METHOD PROTECTED getValue : BOOL //Return value = TRUE if execution finished and state incremented 
VAR_INPUT
	Index						:	WORD;
	SubIndex					:	BYTE;
	Len							:	UDINT;
	pActValue					:	PVOID; //Address of variable for actual value
	pSetValue					:	PVOID; //Address of variable for ser value variable, can be zero if no corresponding SetVariable exists
	CompleteAccess				:	BOOL;
END_VAR
CoERead(bExecute := TRUE , nIndex := Index ,nSubIndex := SubIndex ,pDstBuf := pActValue ,cbBufLen := Len, bCompleteAccess  := CompleteAccess);
IF NOT CoERead.bBUSY 	
THEN
	IF NOT CoERead.bError
	THEN
		IF pSetValue <> 0 THEN MEMCPY(pSetValue, pActValue, Len); END_IF
		state 												:= state + 1; 
	ELSE
		Busy												:= FALSE;
		Error												:= TRUE;
		ErrorId												:= CoERead.nErrId;
		ErrorText											:= CONCAT('Error read parameter in state:' , TO_STRING(state * -1));
		ErrorText											:= CONCAT(ErrorText , ' Id:');
		ErrorText											:= CONCAT(ErrorText , TO_STRING(ErrorId));
		State												:= 9999;
	END_IF
	CoERead(bExecute := FALSE);
	getValue												:= TRUE;
END_IF
END_METHOD

METHOD PROTECTED seqRead : BOOL //Return value = TRUE if execution finished 
VAR_IN_OUT
	State							:	INT;
END_VAR

(* Sequence read parameter **********************************)
	CASE state OF
	1..99: //Read application specific parameter  
		seqRead												:= TRUE;
		
	1001: (* Init step ******************************************************)
		CoERead(bExecute := FALSE, sNetId:= F_CreateAmsNetId(nIds := AdsAddr.netId), nSlaveAddr:= AdsAddr.port);
		IF NOT CoERead.bBusy
		THEN
			state											:= state + 1;	
		END_IF
		
	1002: (* Device name *************************************************************************************)
		IF LEN(DeviceType) > 0 AND NOT CoERead.bBusy
		THEN
			state											:= state + 1;
		ELSE
			getValue(Index:= 16#1008,	Subindex := 16#0,	LEN := SIZEOF(DeviceType),	pActValue := ADR(DeviceType),	pSetValue := 0, completeAccess := FALSE);
		END_IF

			
	1003: (* kp_current *************************************************************************************)
		IF DeviceType = 'EL7041-1000' OR DeviceType = 'EP7041-3002' OR DeviceType = 'EP7041-3102'
		THEN
			state											:= state + 1; (* NOT available *)
		ELSE	
			IF getValue(Index:= 16#8011,	Subindex := 16#01,	LEN := SIZEOF(_UINT),	pActValue := ADR(_UINT),	pSetValue := 0, completeAccess := FALSE)
			THEN
				KpCurrent := SetKpCurrent					:= SEL(Error, UINT_TO_LREAL(_UINT), 0.0);
			END_IF
		END_IF
		
	1004: (* ki current **********************************)
		IF DeviceType = 'EL7041-1000' OR DeviceType = 'EP7041-3002' OR DeviceType = 'EP7041-3102'
		THEN
			state											:= state + 1; (* Not available *)
		ELSE	
			IF getValue(Index:= 16#8011,	Subindex := 16#02,	LEN := SIZEOF(_UINT),	pActValue := ADR(_UINT),	pSetValue := 0, completeAccess := FALSE)
			THEN
				KiCurrent := SetKiCurrent					:= SEL(Error, UINT_TO_LREAL(_UINT), 0.0);
			END_IF		
		END_IF
	
	1005: (* Kp velocity ****************************************************************************************)
		IF DeviceType = 'EL7041-1000'
		THEN
			state											:= state + 1;
		ELSIF DeviceType = 'EL7037' OR DeviceType = 'EL7047' 
		THEN			
			IF getValue(Index:= 16#8014,	Subindex := 16#03,	LEN := SIZEOF(_UDINT),	pActValue := ADR(_UDINT),	pSetValue := 0, completeAccess := FALSE)
			THEN
				KpVelocity := SetKpVelocity					:= SEL(Error, UDINT_TO_LREAL(_UDINT), 0.0);
			END_IF
		ELSE			
			IF getValue(Index:= 16#8013,	Subindex := 16#01,	LEN := SIZEOF(_UINT),	pActValue := ADR(_UINT),	pSetValue := 0, completeAccess := FALSE)
			THEN
				KpVelocity := SetKpVelocity					:= SEL(Error, UINT_TO_LREAL(_UINT), 0.0);
			END_IF			
		END_IF	
		
	1006: (* Tn velocity or Ki Velocity ****************************************************************************************)
		IF DeviceType = 'EL7041-1000'
		THEN
			state											:= state + 1;
		ELSIF DeviceType = 'EL7037' OR DeviceType = 'EL7047'
		THEN (* Tn velocity*)			
			IF getValue(Index:= 16#8014,	Subindex := 16#04,	LEN := SIZEOF(_UINT),	pActValue := ADR(_UINT),	pSetValue := 0, completeAccess := FALSE)
			THEN
				KiVelocity := SetKiVelocity					:= SEL(Error, UINT_TO_LREAL(_UINT), 0.0);
			END_IF
			
		ELSE (* Ki Velccity*)
			IF getValue(Index:= 16#8013,	Subindex := 16#02,	LEN := SIZEOF(_UINT),	pActValue := ADR(_UINT),	pSetValue := 0, completeAccess := FALSE)
			THEN
				KiVelocity := SetKiVelocity					:= SEL(Error, UINT_TO_LREAL(_UINT), 0.0);
			END_IF
		END_IF 
	
	1007: (* Kp position ****************************************************************************************)
		IF DeviceType = 'EL7037' OR DeviceType = 'EL7047' 
		THEN			
			IF getValue(Index:= 16#8014,	Subindex := 16#02,	LEN := SIZEOF(_UINT),	pActValue := ADR(_UINT),	pSetValue := 0, completeAccess := FALSE)
			THEN
				KpPosition := SetKpPosition					:= SEL(Error, UINT_TO_LREAL(_UINT), 0.0);
			END_IF			
		ELSE
			;
		END_IF	
	
	1008: (* Homing cam search direction ****************************************************************************************)		
		IF DeviceType = 'EL7041-1000' 
		THEN
			state											:= state + 1;
		ELSE
			getValue(Index:= 16#8021,	Subindex := 16#13,	LEN := SIZEOF(CalibrInvertDirForCamSearch),	pActValue := ADR(CalibrInvertDirForCamSearch),	pSetValue := ADR(SetCalibrInvertDirForCamSearch), completeAccess := FALSE);			
		END_IF
	
	1009: (* Homing cam of direxction ****************************************************************************************)	
		IF DeviceType = 'EL7041-1000'
		THEN
			state											:= state + 1;
		ELSE
			getValue(Index:= 16#8021,	Subindex := 16#14,	LEN := SIZEOF(CalibrInvertDirForOfCam),	pActValue := ADR(CalibrInvertDirForOfCam),	pSetValue := ADR(SetCalibrInvertDirForOfCam), completeAccess := FALSE);			
		END_IF

	1010: (* Calibration value ****************************************************************************************)
		IF DeviceType = 'EL7041-1000'
		THEN
			state											:= state + 1;
		ELSE
			getValue(Index:= 16#8020,	Subindex := 16#08,	LEN := SIZEOF(CalibrPosition),	pActValue := ADR(CalibrPosition),	pSetValue := ADR(SetCalibrPosition), completeAccess := FALSE);			
		END_IF
		
	ELSE
		state												:= 1;
	END_CASE

(***********************************************************************************)
END_METHOD

METHOD PROTECTED seqWrite : BOOL //Return value = TRUE if execution finished 
VAR_IN_OUT
	State							:	INT;
END_VAR

(* Sequence write parameter *********************************************)
	CASE state OF
	1..99: //Write application specific parameter  
		seqWrite											:= TRUE;
		
	1001: (* Init step ******************************************************)
		CoEWrite(bExecute := FALSE, sNetId:= F_CreateAmsNetId(nIds := AdsAddr.netId), nSlaveAddr:= AdsAddr.port);
		IF NOT CoEWrite.bBusy
		THEN
			state											:= state + 1;	
		END_IF
		
	1002: (* Kv position *************************************************************************************)
		IF DeviceType = 'EL7041-1000' OR DeviceType = 'EP7041-3002' OR DeviceType = 'EP7041-3102'
			OR KpCurrent = SetKpCurrent AND NOT CoEWrite.bBusy
		THEN
			state											:= state + 1;
		ELSE
			_UINT											:= LREAL_TO_UINT(SetKpCurrent);
			IF setValue(Index:= 16#8011,	Subindex := 16#01,	LEN := SIZEOF(_UINT),		pActValue := 0,		pSetValue := ADR(_UINT) , completeAccess := FALSE)
			THEN
				KpCurrent									:= SetKpCurrent;
			END_IF			
		END_IF	
		
	1003: (* ki current **********************************)
		IF DeviceType = 'EL7041-1000' OR DeviceType = 'EP7041-3002' OR DeviceType = 'EP7041-3102'
			OR KiCurrent = SetKiCurrent AND NOT CoEWrite.bBusy
		THEN
			state											:= state + 1;
		ELSE
			_UINT											:= LREAL_TO_UINT(SetKiCurrent);
			IF setValue(Index:= 16#8011,	Subindex := 16#02,	LEN := SIZEOF(_UINT),		pActValue := 0,		pSetValue := ADR(_UINT) , completeAccess := FALSE)
			THEN
				KiCurrent									:= SetKiCurrent;
			END_IF			
		END_IF
	
	1004: (* Kp velocity ****************************************************************************************)
		IF DeviceType = 'EL7041-1000' 
			OR KpVelocity = SetKpVelocity AND NOT CoEWrite.bBusy
		THEN
			state											:= state + 1;
		ELSE
			IF DeviceType = 'EL7037' OR DeviceType = 'EL7047' 
			THEN
				_UDINT										:=LREAL_TO_UDINT(SetKpVelocity);
				IF setValue(Index:= 16#8014,	Subindex := 16#03,	LEN := SIZEOF(_UDINT),		pActValue := 0,		pSetValue := ADR(_UDINT) , completeAccess := FALSE)
				THEN
					KpVelocity								:= SetKpVelocity;
				END_IF	
			ELSE
				_UINT										:=LREAL_TO_UINT(SetKpVelocity);
				IF setValue(Index:= 16#8013,	Subindex := 16#01,	LEN := SIZEOF(_UINT),		pActValue := 0,		pSetValue := ADR(_UINT) , completeAccess := FALSE)
				THEN
					KpVelocity								:= SetKpVelocity;
				END_IF	
			END_IF		
		END_IF
	
	1005: (* Tn velocity or Ki velocity****************************************************************************************)
		IF SetTnVelocity = TnVelocity AND SetKiVelocity = KiVelocity AND NOT CoEWrite.bBusy OR DeviceType = 'EL7041-1000'
		THEN 
			state											:= state + 1;
		ELSE
			IF DeviceType = 'EL7037' OR DeviceType = 'EL7047' 
			THEN (* Tn Velocity *)
				_UINT										:= LREAL_TO_UINT(SetTnVelocity);
				IF setValue(Index:= 16#8014,	Subindex := 16#04,	LEN := SIZEOF(_UINT),		pActValue := 0,		pSetValue := ADR(_UINT) , completeAccess := FALSE)
				THEN
					TnVelocity								:= SetTnVelocity;
				END_IF	
				
	
			ELSE (* Ki Velocity *)
				_UINT										:= LREAL_TO_UINT(SetKiVelocity);
				IF setValue(Index:= 16#8013,	Subindex := 16#02,	LEN := SIZEOF(_UINT),		pActValue := 0,		pSetValue := ADR(_UINT) , completeAccess := FALSE)
				THEN
					KiVelocity								:= SetKiVelocity;
				END_IF				
			END_IF	
		END_IF
	
	1006: (* Kp position ****************************************************************************************)		
		IF SetKpPosition <> KpPosition AND (DeviceType = 'EL7037' OR DeviceType = 'EL7047')
		THEN
			_UINT											:= LREAL_TO_UINT(SetKpPosition);
			IF setValue(Index:= 16#8014,	Subindex := 16#02,	LEN := SIZEOF(_UINT),		pActValue := 0 ,		pSetValue := ADR(_UINT) , completeAccess := FALSE)	
			THEN
				KpPosition									:= SetKpPosition;
			END_IF			
		ELSIF NOT CoEWrite.bBusy
		THEN
			state											:= state + 1;
		END_IF
			
	1007: (* Homing cam search direction ********************************************************************************************)
		IF DeviceType = 'EL7041-1000' 
		THEN
			state											:= state + 1;
		ELSE
			setValue(Index:= 16#8021,	Subindex := 16#13,	LEN := SIZEOF(SetCalibrInvertDirForCamSearch),		pActValue := ADR(CalibrInvertDirForCamSearch) ,		pSetValue := ADR(SetCalibrInvertDirForCamSearch) , completeAccess := FALSE);
		END_IF
		
	1008: (* Homing cam of direction *****************************************************************************************)
		IF DeviceType = 'EL7041-1000' 
		THEN
			state											:= state + 1;
		ELSE
			setValue(Index:= 16#8021,	Subindex := 16#14,	LEN := SIZEOF(SetCalibrInvertDirForOfCam),		pActValue := ADR(CalibrInvertDirForOfCam) ,		pSetValue := ADR(SetCalibrInvertDirForOfCam) , completeAccess := FALSE)	;	
		END_IF
	
	1009: (* Calibration position ***********************************************************************)	
		IF DeviceType = 'EL7041-1000' 
		THEN
			state											:= state + 1;
		ELSE
			setValue(Index:= 16#8020,	Subindex := 16#08,	LEN := SIZEOF(SetCalibrPosition),		pActValue := ADR(CalibrPosition) ,		pSetValue := ADR(SetCalibrPosition) , completeAccess := FALSE)	;	
		END_IF
	ELSE
		state												:= 1;
	END_CASE

(************************************************************************************)
END_METHOD

METHOD PROTECTED setValue : BOOL //Return value = TRUE if execution finished and state incremented 
VAR_INPUT
	Index						:	Word;
	SubIndex					:	BYTE;
	Len							:	UDINT;
	pActValue					:	PVOID; //Address of variable for actual value, can be zero if no corresponding acual value variable exists
	pSetValue					:	PVOID; //Address of variable for set value variable
	CompleteAccess				:	BOOL;
END_VAR


IF pActValue <> 0 AND pSetValue <> 0 AND_THEN MEMCMP(pSetValue, pActValue, Len) = 0
THEN //Skip write parameter if set and actual value are equel
	state													:= state + 1;	
	setValue												:= TRUE;
ELSE
	CoEWrite(bExecute := TRUE, nIndex := Index ,nSubIndex := SubIndex , pSrcBuf := pSetValue ,cbBufLen := Len , bCompleteAccess := CompleteAccess );
	IF NOT CoEWrite.bBusy
	THEN
		IF NOT CoEWrite.bError
		THEN
			IF pActValue <> 0 THEN MEMCPY(pActValue, pSetValue, Len); END_IF	
			state											:= state + 1;
		ELSE
			Busy											:= FALSE;
			Error											:= TRUE;
			ErrorId											:= CoEWrite.nErrId;
			ErrorText										:= CONCAT('Error write parameter in state:' , TO_STRING(state * -1));
			ErrorText										:= CONCAT(ErrorText , ' Id:');
			ErrorText										:= CONCAT(ErrorText , TO_STRING(ErrorId));
			State											:= 9999;
		END_IF
		CoEWrite(bExecute := FALSE);
		setValue											:= TRUE;
	END_IF		
END_IF
END_METHOD

END_FUNCTION_BLOCK

// POUs/IO/Drives/AxDriveGetRef
{attribute 'no_check'}
//Provides drive reference (Ref -> ST_DriveRef) based on NC-AxisID
//Drive reference is needed for FB's of lib Drive e.g. FB_SoEAX5000FirmwareUpdate_ByDriveRef
FUNCTION_BLOCK AxDriveGetRef EXTENDS FbBase
VAR CONSTANT                								
	NCIDXG_AXPARMS											: UDINT := 16#0000_4000;	(* Axis with ID: Parameter 			*)
	NCIDXO_AXP_HWAMSADDR									: UDINT := 16#0000_0031;	
	MIN_ADSREAD_BUFFER										:	INT := 0;
	MAX_ADSREAD_BUFFER										:	INT := 9;
END_VAR 
VAR_INPUT                   					
	AmsNetId												: T_AmsNetId := '';	(* netID of PC with NC *)			      
	AxisId													:	DWORD; //NC axis id	
END_VAR
VAR_OUTPUT                  								
	DriveAmsNetId											: T_AmsNetIdArr; (* Ams net id as array of bytes *)
    DriveRef												: ST_DriveRef; 	(* contains sNetID of EcMaster, nSlaveAddr of EcDrive, nDriveNo of EcDrive, either preset or read from NC *)
END_VAR              								                 								
VAR                         								
(* cache ********************************************)
	AdsReadBuffer											: ARRAY[MIN_ADSREAD_BUFFER..MAX_ADSREAD_BUFFER] OF BYTE;
                						
(* trigger ******************************************)

(* timer ********************************************)
	
(* blocks *******************************************)	
	AdsRead													: ADSREAD := (TMOUT := DEFAULT_ADS_TIMEOUT);
	
(* dummys *******************************************)
END_VAR

	(* Create drive ref for device 									*)
	(****************************************************************)

(* Sequence ****************************************)
	rtExecute(CLK := Execute);
	CASE state OF 
	0:	
		Busy												:= FALSE;
		IF NOT Execute
		THEN
			Done											:= FALSE;
			Error											:= FALSE;
			ErrorId											:= 0;
		ELSIF rtExecute.Q
		THEN
			Busy											:= TRUE;
			Done											:= FALSE;
			Error											:= FALSE;
			ErrorId											:= 0;
			AdsRead(READ := FALSE);
			MEMSET(ADR(DriveRef), 0, SIZEOF(DriveRef));
			MEMSET(ADR(AdsReadBuffer), 0, SIZEOF(AdsReadBuffer));
			state											:= State + 1;
		END_IF 
	
	1: //Get drive slave address
		AdsRead(
			NETID	:= AmsNetId,
			PORT	:= AMSPORT_R0_NC,
			IDXGRP	:= NCIDXG_AXPARMS + AxisId,
			IDXOFFS	:= NCIDXO_AXP_HWAMSADDR,
			LEN		:= SIZEOF(AdsReadBuffer) ,
			DESTADDR:= ADR(AdsReadBuffer),
			READ	:= TRUE);
		IF NOT AdsRead.BUSY
		THEN
			IF NOT AdsRead.ERR 
			THEN
				MEMCPY(ADR(DriveAmsNetId), ADR(AdsReadBuffer), SIZEOF(DriveAmsNetId)); 							(* AdsreadBuffer[0..5] *)
				MEMCPY(ADR(DriveRef.nSlaveAddr), ADR(AdsReadBuffer[6]), SIZEOF(DriveRef.nSlaveAddr));  	(* AdsreadBuffer[6..7] *)
				MEMCPY(ADR(DriveRef.nDriveNo), ADR(AdsReadBuffer[8]), SIZEOF(DriveRef.nDriveNo));  		(* AdsreadBuffer[8..9] *)

				(* create string out of byte array *)
				DriveRef.sNetId 							:= F_CreateAmsNetId(DriveAmsNetId);
				
				Busy										:= FALSE;
				Done										:= TRUE;
				state										:= 0;
			ELSE
				Busy										:= FALSE;
				Error										:= TRUE;
				ErrorId										:= AdsRead.ERRID;
				State										:= 0;
			END_IF
		END_IF
	END_CASE
	
(**********************************************************************************)

END_FUNCTION_BLOCK

// POUs/IO/EL-EP/EL3403/EL3403
{attribute 'no_check'}
FUNCTION_BLOCK EL3403 Extends EcSlaveInfoData
VAR CONSTANT
	MIN_PHASE												:	INT := 1;
	MAX_PHASE												:	INT := 3;
END_VAR  
VAR_INPUT
	IndexOut										AT %Q*	:	ARRAY[MIN_PHASE..MAX_PHASE] OF USINT;
	Transmission											:	ARRAY[MIN_PHASE..MAX_PHASE] OF LREAL;	//Transmission current transformator for each phase e.g. 750 *)
END_VAR
VAR_OUTPUT
	(* Inputs Channel 1-3 *)
	TxPDOToggle										AT %I*	: 	ARRAY[MIN_PHASE..MAX_PHASE] OF BOOL;
	IndexIn											AT %I*	: 	ARRAY[MIN_PHASE..MAX_PHASE] OF USINT;
	Current													: 	ARRAY[MIN_PHASE..MAX_PHASE] OF LREAL; 	//Unit: 0,000001 A
	Voltage													: 	ARRAY[MIN_PHASE..MAX_PHASE] OF LREAL; 	//Unit: 0,0001 V
	ActivePower												: 	ARRAY[MIN_PHASE..MAX_PHASE] OF LREAL; 	//Unit: 0,01 W

	(* PM Status Data *)
	MissingZeroCrossingA							AT %I*	: 	BOOL;
	MissingZeroCrossingB							AT %I* 	: 	BOOL;
	MissingZeroCrossingC							AT %I* 	: 	BOOL;
	PhaseSequenceError								AT %I* 	: 	BOOL;
//	SyncError										AT %I* 	: 	BOOL;
                                                              	
	(* MultiplexValues	*)
	ApparentPower											:	ARRAY[MIN_PHASE..MAX_PHASE] OF LREAL; 	//apparent power unit: 0,01 VA
	ReactivePower											:	ARRAY[MIN_PHASE..MAX_PHASE] OF LREAL; 	//reactive power unit: 0,01 VAr
	PowerFactor												:	ARRAY[MIN_PHASE..MAX_PHASE] OF LREAL; 	//effective power cos phi Unit: 0,001
	EnergyConsumption										:	ARRAY[MIN_PHASE..MAX_PHASE] OF LREAL; 	//energy unit: 0,001 Wh
	EnergyConsumptionInvers									:	ARRAY[MIN_PHASE..MAX_PHASE] OF LREAL; 	//energy unit: 0,001 Wh
	TimestampDistClocks										:	ARRAY[MIN_PHASE..MAX_PHASE] OF LREAL; 	//timestamp unit : 1 ns
	Frequency												:	ARRAY[MIN_PHASE..MAX_PHASE] OF LREAL; 	//frequenzy unit : 0,1 Hz

END_VAR
VAR (* Internal IOs *)
	_Current										AT %I* 	: 	ARRAY[MIN_PHASE..MAX_PHASE] OF DINT; 	//Unit: 0,000001 A
	_Voltage										AT %I* 	: 	ARRAY[MIN_PHASE..MAX_PHASE] OF DINT; 	//Unit: 0,0001 V
	_ActivePower									AT %I* 	: 	ARRAY[MIN_PHASE..MAX_PHASE] OF DINT; 	//Unit: 0,01 W

	_VariantValue									AT %I* 	: 	ARRAY[MIN_PHASE..MAX_PHASE] OF DINT;
//	_SyncErrorChannel								AT %I* 	: 	ARRAY[MIN_PHASE..MAX_PHASE] OF BOOL; 	//reserved
//	_SyncErrorTerminal										: 	BOOL;	//reserved
END_VAR                       							
VAR
	i														:	INT;
END_VAR

(* EL 3403 IO 									*)
(************************************************)

(* Get Index Values *****************************)
	FOR i := MIN_PHASE TO MAX_PHASE DO
		Current[i]											:= Transmission[i] * DINT_TO_LREAL(_Current[i]) / 1000000.0; //A
		Voltage[i]											:= (*Uebersetzung[i] **) DINT_TO_LREAL(_Voltage[i]) / 10000.0; //V
		ActivePower[i]										:= Transmission[i] * DINT_TO_LREAL(_ActivePower[i]) / 100.0; //W
                                            				
		CASE IndexIn[i] OF                  				
		0:(*Scheinleistung*)                				
			ApparentPower[i]								:= Transmission[i] * DINT_TO_LREAL(_VariantValue[i]) / 100.0; //VA
                                            				
		1:(*Blindleistung*)                 				
			ReactivePower[i]								:= Transmission[i] * DINT_TO_LREAL(_VariantValue[i]) / 100.0; //VAr
                                            				
		2:(*Energie*)                       				
			EnergyConsumption[i]							:= Transmission[i] * DINT_TO_LREAL(_VariantValue[i]) / 1000.0; //Wh
                                            				
		3:(*Wirkleistungsfaktor*)           				
			PowerFactor[i]									:= DINT_TO_LREAL(_VariantValue[i]) / 1000.0; //cos phi
                                            				
		4:(*Frequenz*)                      	
			Frequency[i]									:= DINT_TO_LREAL(_VariantValue[i]) / 10.0; //Hz
                                            				
		5:(*Energie Invers*)                				
			EnergyConsumptionInvers[i]						:= Transmission[i] * DINT_TO_LREAL(_VariantValue[i]) / 1000.0;
                                            				
		100:(*Zeitstempel*)                 				
			TimestampDistClocks[i]							:= DINT_TO_LREAL(_VariantValue[i]);
	
		END_CASE

	END_FOR

(***********************************************)

END_FUNCTION_BLOCK

// POUs/IO/EL-EP/EL3403/EL3403Logic
{attribute 'no_check'}
//FB gets raw data from EL3404 every cycle and calculate real values *)
FUNCTION_BLOCK EL3403Logic
VAR_INPUT
	TrigReadVariantValues									:	BOOL 	:= FALSE;	//Rising edge reports actual total values on FB outputs
	Transmission											:	LREAL 	:= 750.0; 	//Transmission current transformator
	Mode													:	INT 	:= 0; 		(* 	0 = Phase 1-3
																					  	1 = Phase 1
																					 	2 = Phase 2
																					 	3 = Phase 3 *)                                   						
END_VAR                             	
VAR_OUTPUT
	(* Components OUTPUT -> ReadOnly ! *)
	IO														:	EL3403;
                                    				                                					
	(* Total Values *)              					
	TotalEffectivePower										: 	LREAL; 	//W
	TotalPowerFactor										: 	LREAL; 	//total power factor cos phi
	TotalEnergyConsumption									: 	LREAL; 	//Wh
                                    					
	(* Error *)                     					
	ErrorPhaseSequence										:	BOOL;
	ErrorMissingZeroCrossing								:	BOOL;
	TimeStart												: 	TIME;		(* Startzeit *)
	TimeEnd													: 	TIME;		(* Endzeit *)
	TimeDiff												: 	TIME;		(* Differenz Start End *)
	
	(* Ctrl Status  *)              					
	Valid													:	BOOL;	//TRUE when data is valid
	Busy													:	BOOL;	//Busy is TRUE at the rising edge of Execute and FALSE when one of the outputs Done, Aborted, or Error is set 
	Error													:	BOOL;	//Rising edge of Error informs that an error occurred during the execution of the Function Block 

END_VAR                             	
VAR                                 	
	rtReadVariantValues										:	R_Trig;
	state													:	INT;
	_MIN_PHASE												:	INT;
	_MAX_PHASE												:	INT;
	i														:	INT;
END_VAR

(* Work EL3403 data 						*)
(********************************************)

(* Work Termianl IO ******************************************)
	FOR i := IO.MIN_PHASE TO IO.MAX_PHASE 
	DO
		IO.Transmission[i] 									:= Transmission;
	END_FOR

	IO();

(* Error *****************************************************)
	Error 													:= IO.WCState OR IO.InfoDataState <> Tc2_EtherCAT.EC_DEVICE_STATE_OP;

(* Get Total Values ******************************************)
IF NOT Error
THEN
	CASE Mode OF
	1:
		TotalEffectivePower 								:= IO.ActivePower[1];
		TotalPowerFactor 									:= IO.PowerFactor[1];
		TotalEnergyConsumption 								:= IO.EnergyConsumption[1];
	2:                              						
		TotalEffectivePower 								:= IO.ActivePower[2];
		TotalPowerFactor 									:= IO.PowerFactor[2];
		TotalEnergyConsumption 								:= IO.EnergyConsumption[2];
	3:                              						
		TotalEffectivePower 								:= IO.ActivePower[3];
		TotalPowerFactor 									:= IO.PowerFactor[3];
		TotalEnergyConsumption 								:= IO.EnergyConsumption[3];
	ELSE (* Phase 1-3 *)            						
		TotalEffectivePower 								:= IO.ActivePower[1] + IO.ActivePower[2] + IO.ActivePower[3];
		TotalPowerFactor 									:= (IO.PowerFactor[1] + IO.PowerFactor[2] + IO.PowerFactor[3]) / 3.0;
		TotalEnergyConsumption 								:= IO.EnergyConsumption[1] + IO.EnergyConsumption[2] + IO.EnergyConsumption[3];
	END_CASE                        	

END_IF

(* Trigger ReadVariantValues ******************************)
rtReadVariantValues(CLK := TrigReadVariantValues);

IF rtReadVariantValues.Q
	OR state <> 0
THEN
	ReadVariantValues(Mode := Mode);
END_IF

(********************************************************)

METHOD PUBLIC readVariantValues : Bool //Return value = TRUE if busy
VAR_INPUT
	Mode								:	INT 	:= 0; (* 	0 = Phase 1-3
															  		1 = Phase 1
															 	 	2 = Phase 2
															 		3 = Phase 3 *)
END_VAR
IF state = 0 
THEN
	THIS^.Mode												:= Mode;
	CASE mode OF
	1:
		_MIN_PHASE 											:= IO.MIN_PHASE;
		_MAX_PHASE 											:= IO.MIN_PHASE;
	2:             											
		_MIN_PHASE 											:= IO.MIN_PHASE + 1;
		_MAX_PHASE 											:= IO.MIN_PHASE + 1;
	3:             											
		_MIN_PHASE 											:= IO.MAX_PHASE;
		_MAX_PHASE 											:= IO.MAX_PHASE;
	ELSE           											
		_MIN_PHASE 											:= IO.MIN_PHASE;
		_MAX_PHASE 											:= IO.MAX_PHASE;
	END_CASE
	state 													:= 1;
	TimeStart 												:= TIME();
END_IF

(* Read Variant Values *******************************)
	CASE state OF
	0:
		;
		
	1:
		FOR i := _MIN_PHASE TO _MAX_PHASE DO
			IO.IndexOut[i] 									:= 0;
			IF IO.IndexIn[i] = IO.IndexOut[i]
				AND i = _MAX_PHASE
			THEN (* Set Next index *)
				state 										:= 2;
			ELSE
				;
			END_IF
		END_FOR

	2:
		FOR i := _MIN_PHASE TO _MAX_PHASE DO
			IO.IndexOut[i] 									:= 1;
			IF IO.IndexIn[i] = IO.IndexOut[i]
				AND i = _MAX_PHASE
			THEN (* Set Next index *)
				state 										:= 3;
			ELSE
				;
			END_IF
		END_FOR
	3:
		FOR i := _MIN_PHASE TO _MAX_PHASE DO
			IO.IndexOut[i] 									:= 2;
			IF IO.IndexIn[i] = IO.IndexOut[i]
				AND i = _MAX_PHASE
			THEN (* Set Next index *)
				state 										:= 4;
			ELSE
				;
			END_IF
		END_FOR
	4:
		FOR i := _MIN_PHASE TO _MAX_PHASE DO
			IO.IndexOut[i] 									:= 3;
			IF IO.IndexIn[i] = IO.IndexOut[i]
				AND i = _MAX_PHASE
			THEN (* Set Next index *)
				state 										:= 5;
			ELSE
				;
			END_IF
		END_FOR
	5:
		FOR i := _MIN_PHASE TO _MAX_PHASE DO
			IO.IndexOut[i] 									:= 4;
			IF IO.IndexIn[i] = IO.IndexOut[i]
				AND i = _MAX_PHASE
			THEN (* Set Next index *)
				state 										:= 6;
			ELSE
				;
			END_IF
		END_FOR

	6:
		FOR i := _MIN_PHASE TO _MAX_PHASE DO
			IO.IndexOut[i] 									:= 5;
			IF IO.IndexIn[i] = IO.IndexOut[i]
				AND i = _MAX_PHASE
			THEN (* Set Next index *)
				state 										:= 7;
			ELSE
				;
			END_IF
		END_FOR

	7:
		FOR i := _MIN_PHASE TO _MAX_PHASE DO
			IO.IndexOut[i] 									:= 100;
			IF IO.IndexIn[i] = IO.IndexOut[i]
				AND i = _MAX_PHASE
			THEN (* Set Next index *)
				Valid 										:= TRUE;
				state 										:= 0;
				TimeEnd 									:= TIME();
				TimeDiff 									:= TimeEnd - TimeStart;
			ELSE
				;
			END_IF
		END_FOR

	END_CASE
	
	Busy													:= state <> 0;
	ReadVariantValues 										:= Busy;
END_METHOD

END_FUNCTION_BLOCK

// POUs/IO/EL-EP/EL9x/EL95xxPowerTerminal
{attribute 'no_check'}
FUNCTION_BLOCK EL95xxPowerTerminal 
VAR_OUTPUT CONSTANT
END_VAR
VAR_INPUT
END_VAR
VAR_OUTPUT	
	PowerOK			 									AT  %I* : BOOL;
	Overload											AT  %I* : BOOL;
END_VAR
VAR
END_VAR

	(* EL95xx Power supply terminal			*)
	(****************************************)
	
(* Work objects ****************************************)
;
(*******************************************************)

END_FUNCTION_BLOCK

// POUs/IO/EL-EP/EL9x/ELSystemTerminal
{attribute 'no_check'}
FUNCTION_BLOCK ELSystemTerminal //e.g. EL9410
VAR_OUTPUT CONSTANT
END_VAR
VAR_INPUT
END_VAR
VAR_OUTPUT	
	UsUndervoltage		 								AT  %I* : BOOL;
	UpUndervoltage										AT  %I* : BOOL;
END_VAR
VAR
END_VAR

	(* System terminal power status			*)
	(****************************************)
	
(* Work objects ****************************************)
;
(*******************************************************)

END_FUNCTION_BLOCK

// POUs/IO/EL-EP/EP92xxPwrBox/EP9214
{attribute 'no_check'}
FUNCTION_BLOCK EP9214
VAR_OUTPUT CONSTANT
	MIN_CHANNEL												: INT := 1;
	MAX_CHANNEL												: INT := 4;
END_VAR
VAR_INPUT
	EnableControlViaFieldbus					AT  %Q* 	: 	BOOL := FALSE;	//FB will be processed as long as enable is TRUE
	ResetTrig									AT  %Q* 	: 	BOOL := FALSE;	//The box will be reseted with a rising edge 
	
	Channel													:	ARRAY[MIN_CHANNEL..MAX_CHANNEL] OF EP9214_CHANNEL;
END_VAR     								
VAR_OUTPUT  	
	TempWarning									AT  %I* 	: 	BOOL;	//TRUE when temperature warning occurs
	TempError									AT  %I* 	: 	BOOL;	//TRUE when temperature error occurs
	UsWarning									AT  %I* 	: 	BOOL;	//TRUE when system voltage warning occurs
	UsError										AT  %I* 	: 	BOOL;	//TRUE when system voltage error occurs
	UpWarning									AT  %I* 	: 	BOOL;	//TRUE when peripheral voltage warning occurs
	UpError										AT  %I* 	: 	BOOL;	//TRUE when peripheral voltage error occurs
	GlobalError									AT  %I* 	: 	BOOL;	//TRUE when global error occurs
	ResetInput									AT  %I* 	: 	BOOL;	//Resets box with a rising edge
	TxPDOState									AT  %I* 	: 	BOOL;	
	TxPDOToggle									AT  %I* 	: 	BOOL;	
END_VAR     								
VAR
	i														:	INT;
END_VAR

;

{attribute 'monitoring' := 'call'}
PROPERTY PUBLIC channelErrorUp : int
GET
ChannelErrorUp				:= 0;
FOR i := MIN_CHANNEL TO MAX_CHANNEL do
	IF Channel[i].ErrorUp
	THEN
		ChannelErrorUp			:= i;
		EXIT;
	END_IF	
END_FOR
END_GET
END_PROPERTY

{attribute 'monitoring' := 'call'}
PROPERTY PUBLIC channelErrorUs : int
GET
ChannelErrorUs				:= 0;
FOR i := MIN_CHANNEL TO MAX_CHANNEL do
	IF Channel[i].ErrorUs
	THEN
		ChannelErrorUs			:= i;
		EXIT;
	END_IF	
END_FOR
END_GET
END_PROPERTY

{attribute 'monitoring' := 'call'}
PROPERTY PUBLIC channelWarningUp : int
GET
ChannelWarningUp					:= 0;
FOR i := MIN_CHANNEL TO MAX_CHANNEL do
	IF Channel[i].WarningUp	
	THEN
		ChannelWarningUp			:= i;
		EXIT;
	END_IF	
END_FOR
END_GET
END_PROPERTY

{attribute 'monitoring' := 'call'}
PROPERTY PUBLIC channelWarningUs : int
GET
ChannelWarningUs					:= 0;
FOR i := MIN_CHANNEL TO MAX_CHANNEL do
	IF Channel[i].WarningUs	
	THEN
		ChannelWarningUs			:= i;
		EXIT;
	END_IF	
END_FOR
END_GET
END_PROPERTY

END_FUNCTION_BLOCK

// POUs/IO/EL-EP/EP92xxPwrBox/EP9214_CHANNEL
{attribute 'no_check'}
FUNCTION_BLOCK EP9214_CHANNEL
VAR_INPUT
	EnableUs									AT  %Q* 	: 	BOOL := TRUE; 	//switches system voltage on with a rising edge
	EnableUp									AT  %Q* 	: 	BOOL := TRUE; 	//switches peripheral voltage on with a rising edge
	ResetTrigUs	                                AT  %Q* 	: 	BOOL := FALSE;  //resets system voltage with a rising edge                    
	ResetTrigUp                                 AT  %Q* 	: 	BOOL := FALSE;	//resets peripheral voltage with a rising edge                                                                                           
END_VAR     								                          
VAR_OUTPUT  								                          
	ErrorUs										AT  %I* 	: 	BOOL := FALSE;	//TRUE when system voltage error occurs 
	ErrorUp										AT  %I* 	: 	BOOL := FALSE; 	//TRUE when peripheral voltage error occurs 
	WarningUs									AT  %I* 	: 	BOOL := FALSE; 	//TRUE when system voltage warning occurs 
	WarningUp									AT  %I* 	: 	BOOL := FALSE; 	//TRUE when peripheral voltage warning occurs 
	StatusUs									AT  %I* 	: 	BOOL := FALSE; 	//TRUE when system voltage is on
	StatusUp									AT  %I* 	: 	BOOL := FALSE; 	//TRUE when peripheral voltage is on 
	ChannelError								AT  %I* 	: 	BOOL := FALSE; 	//TRUE when channel error occurs 
	SyncError									AT  %I* 	: 	BOOL := FALSE; 	//TRUE when synchronization error occurs 
	TxPDOState									AT  %I* 	: 	BOOL := FALSE; 
	TxPDOToggle									AT  %I* 	: 	BOOL := FALSE; 
END_VAR     								
VAR
END_VAR

;

END_FUNCTION_BLOCK

// POUs/IO/EL-EP/EP92xxPwrBox/EP9224_0037
FUNCTION_BLOCK EP9224_0037
VAR_OUTPUT CONSTANT
	MIN_CHANNEL												:	INT := 1;
	MAX_CHANNEL												:	INT := 4;
END_VAR
VAR_INPUT
	EnableControlViaFieldbus					AT  %Q* 	: 	BOOL := TRUE;	// FB will be processed ads long as enable is TRUE
	ResetTrig									AT  %Q* 	: 	BOOL := FALSE;	// The box will be reseted with a rising edge 
	
	Channel													:	ARRAY[MIN_CHANNEL..MAX_CHANNEL] OF EP9224_0037_CHANNEL;
END_VAR     								
VAR_OUTPUT  
	CurrentUs									AT	%I*		:	INT;	// Actual Current Us
	CurrentUp									AT	%I*		:	INT;	// Actual Current Up
	VoltageUs									AT 	%I*		:	INT;	// Actual Voltage Us
	VoltageUp									AT 	%I*		:	INT;	// Actual Voltage Up
	Temperature									AT 	%I*		:	INT;	// Actual Temperature
	
	TempWarning												: 	BOOL;	// TRUE when temperature warning occurs
	TempError												: 	BOOL;	// TRUE when temperature error occurs
	UsWarning												: 	BOOL;	// TRUE when system voltage warning occurs
	UsError													: 	BOOL;	// TRUE when system voltage error occurs
	UpWarning												: 	BOOL;	// TRUE when peripheral voltage warning occurs
	UpError													: 	BOOL;	// TRUE when peripheral voltage error occurs
	GlobalError												: 	BOOL;	// TRUE when global error occurs
	SumCurrentWarning										:	BOOL;	// TRUE when Sum Current Warning occurs
	SumCurrentError											:	BOOL;	// True when Sum Current Error occurs
	ResetInput												: 	BOOL;	// Resets box with a rising edge
	TxPDOState												: 	BOOL;	
	TxPDOToggle												: 	BOOL;	
END_VAR     								
VAR
{attribute 'displaymode':='binary'}
	status										AT 	%I*		: 	WORD;	// Statusword
	i														:	INT;
END_VAR

FOR i := MIN_CHANNEL TO MAX_CHANNEL
DO
	Channel[i]();
END_FOR

	TempWarning			     									:= status.0;
	TempError			        								:= status.1;
	UsWarning			       								   	:= status.2;		         	     			 			
	UsError				           								:= status.3;
	UpWarning			             							:= status.4;
	UpError				           								:= status.5;
	GlobalError			    									:= status.6;
	SumCurrentWarning											:= status.7;
	SumCurrentError		     									:= status.8;
	ResetInput			     									:= status.9;
	TxPDOState			     									:= status.10;
	TxPDOToggle													:= status.11;

{attribute 'monitoring' := 'call'}
PROPERTY channelErrorUp : INT
GET
ChannelErrorUp				:= 0;
FOR i := MIN_CHANNEL TO MAX_CHANNEL do
	IF Channel[i].ErrorUp
	THEN
		ChannelErrorUp			:= i;
		EXIT;
	END_IF	
END_FOR
END_GET
END_PROPERTY

{attribute 'monitoring' := 'call'}
PROPERTY channelErrorUs : INT
GET
ChannelErrorUs				:= 0;
FOR i := MIN_CHANNEL TO MAX_CHANNEL do
	IF Channel[i].ErrorUs
	THEN
		ChannelErrorUs			:= i;
		EXIT;
	END_IF	
END_FOR
END_GET
END_PROPERTY

{attribute 'monitoring' := 'call'}
PROPERTY channelWarningUp : INT
GET
ChannelWarningUp					:= 0;
FOR i := MIN_CHANNEL TO MAX_CHANNEL do
	IF Channel[i].WarningUp
	THEN
		ChannelWarningUp			:= i;
		EXIT;
	END_IF	
END_FOR
END_GET
END_PROPERTY

{attribute 'monitoring' := 'call'}
PROPERTY channelWarningUs : INT
GET
ChannelWarningUs					:= 0;
FOR i := MIN_CHANNEL TO MAX_CHANNEL do
	IF Channel[i].WarningUs
	THEN
		ChannelWarningUs			:= i;
		EXIT;
	END_IF	
END_FOR
END_GET
END_PROPERTY

END_FUNCTION_BLOCK

// POUs/IO/EL-EP/EP92xxPwrBox/EP9224_0037_CHANNEL
FUNCTION_BLOCK EP9224_0037_CHANNEL
VAR_INPUT
	OutputUs					AT %Q*	:	BOOL := TRUE;	// switches system voltage on with a rising edge
	OutputUp					AT %Q*	:	BOOL := TRUE;  // resets system voltage with a rising edge      
	ResetTrigUs					AT %Q*	:	BOOL := FALSE;   // switches peripheral voltage on with a rising edge
	ResetTrigUp					AT %Q*	:	BOOL := FALSE;  // resets peripheral voltage with a rising edge        
END_VAR
VAR_OUTPUT	
	CurrentUs					AT %I*	:	INT;			// Actual Us current
	CurrentUp					AT %I*	:	INT;			// Actual Up current
	ErrorUs								:	BOOL := FALSE;	// TRUE when system voltage error occurs 
	ErrorUp								:	BOOL := FALSE; 	// TRUE when peripheral voltage error occurs
	WarningUs							:	BOOL := FALSE; 	// TRUE when system voltage warning occurs 
	WarningUp							:	BOOL := FALSE; 	// TRUE when peripheral voltage warning occurs 
	StatusUs							:	BOOL := FALSE; 	// TRUE when system voltage is on
	StatusUp							:	BOOL := FALSE; 	// TRUE when peripheral voltage is on 
	ChannelError						:	BOOL := FALSE; 	// TRUE when channel error occurs 
	ErrorSumCurrent						:	BOOL;			// TRUE when SumCurrent Error occurs 
	WarningSumCurrent					:	BOOL;			// TRUE when SumCurrent Warning occurs 
	TxPDOState							:	BOOL;
	TxPDOToggle							:	BOOL;
END_VAR
VAR
{attribute 'displaymode':='binary'}
	status						AT %I*	:	WORD;			// Statusword
END_VAR

	
							
	ErrorUs			 					:= status.0;
	ErrorUp             				:= status.1;
	WarningUs            			   	:= status.2;		         	     			 			
	WarningUp		 	    			:= status.3;
	StatusUs 			       			:= status.4;
	StatusUp 		        			:= status.5;
	ChannelError						:= status.6;
	ErrorSumCurrent						:= status.7;
	WarningSumCurrent	    			:= status.8;
	TxPDOState							:= status.9;
	TxPDOToggle							:= status.10;

END_FUNCTION_BLOCK

// POUs/IO/EL-EP/EL1904
{attribute 'no_check'}
FUNCTION_BLOCK EL1904 (* EL Safety Input Terminal IO *)
VAR_INPUT
END_VAR
VAR_OUTPUT
	C1												AT  %I* : BOOL;	//TRUE when channel 1 has high signal
	C2												AT  %I* : BOOL;	//TRUE when channel 2 has high signal
	C3												AT  %I* : BOOL;	//TRUE when channel 3 has high signal
	C4												AT  %I* : BOOL;	//TRUE when channel 4 has high signal
	Valid													: BOOL;	//TRUE when data is valid
END_VAR		            							
VAR                     							
	FSoESlaveCMD									AT  %I* : USINT;
END_VAR

(* EL 1904 Terminal Inputs					             	 V1.2	*)
(********************************************************************)

(* Input Signals Valid ******************************************************)
	Valid 													:= FSoESlaveCMD = 16#36
																	OR FSoESlaveCMD = 16#08;
          													
(**********************************************************************)

END_FUNCTION_BLOCK

// POUs/IO/EL-EP/EL3356
{attribute 'no_check'}
//EL3356 load cell analysis (resistor bridge) process image
//Mode of operation = Standard (Real or INT32)
FUNCTION_BLOCK EL3356 EXTENDS EcSlaveInfoDataExt
VAR_INPUT
//RMB Control
	StartCalib										AT  %Q* : 	BOOL; 
	DisableCalib									AT  %Q* : 	BOOL;
	InputFreeze										AT  %Q* : 	BOOL;
	SampleMode										AT  %Q* : 	BOOL; //1=High speed and low latency / only on EL3356-0010
	Tara											AT  %Q* : 	BOOL;				
END_VAR                     			    					
VAR_OUTPUT                      					
//RMB Status
	Overrange										AT  %I*	:	BOOL;
	DataInvalid										AT  %I*	:	BOOL;
	Error											AT  %I*	:	BOOL;
	CalibInProgress									AT  %I*	:	BOOL;
	SteadyState										AT  %I*	:	BOOL;
	SyncError										AT  %I*	:	BOOL;
	TxPDOToggle										AT  %I* : 	BOOL;
	
//RMB Value
	InReal											AT  %I* : 	REAL; //RMP Value Real 32		
	InInt32											AT  %I* : 	DINT; //RMB Value INT32
END_VAR
VAR
END_VAR

(* EL3356 IOs											             	 		*)
(********************************************************************************)

(* ******************************************************************************)
	;
(********************************************************************************)

{attribute 'monitoring' := 'call'}
PROPERTY PUBLIC inError : BOOL
GET
inError													:= Error OR SyncError OR WcState OR InfoDataState <> Tc2_EtherCAT.EC_DEVICE_STATE_OP;
END_GET
END_PROPERTY

{attribute 'monitoring' := 'call'}
PROPERTY PUBLIC Q : LREAL
GET
IF InInt32 <> 0
THEN
	Q 														:= TO_LREAL(InInt32);
ELSE
	Q 														:= TO_LREAL(InReal);
END_IF
END_GET
END_PROPERTY

END_FUNCTION_BLOCK

// POUs/IO/EL-EP/EL69xx
{attribute 'no_check'}
FUNCTION_BLOCK EL69xx EXTENDS EcSlaveInfoDataExt
VAR_INPUT
(* standard DEVICE Outputs *)
	Control											AT  %Q* : UINT;	
END_VAR                         					
VAR_OUTPUT                      					
(* Device Info Data. Only available if the Checkbox under the register TwinSafe_Logic is selected *)
{attribute 'displaymode':='hex'}
	ProjectCRC 										AT  %I* : UINT;
	SerialNumber									AT  %I* : UDINT;
                                					
(* standard DEVICE Inputs *)    					
	SafetyProjectState								AT  %I* : BYTE; 	//To create the mapping select change Link and select "All Types", then select the variable and press OK
	LoginActive										AT  %I* : BOOL;	
	InputSizeMismatch								AT  %I* : BOOL;
	OutputSizeMismatch								AT  %I* : BOOL;
	TxPDOState										AT  %I* : BOOL;
	TxPDOToggle										AT  %I* : BOOL;	
END_VAR
VAR
END_VAR

Super^(); //Get device name

END_FUNCTION_BLOCK

// POUs/IO/EL-EP/EL9576
{attribute 'no_check'}
//EL Brake Chopper IOs
FUNCTION_BLOCK EL9576 
VAR_OUTPUT CONSTANT
END_VAR
VAR_INPUT
END_VAR
VAR_OUTPUT	
	Overtemperature									AT  %I* : BOOL;		//TRUE when there is an overtemperature on the PCB
	I2T_Error										AT  %I* : BOOL;		//TRUE when there is an overtemperature in the external resistor
	I2T_Warning										AT  %I* : BOOL;		//TRUE when the warning temperature threshold value from the CoE data has been exceeded
	Overvoltage										AT  %I* : BOOL;		//TRUE when the overvoltage threshold value has been exceeded
	Undervoltage									AT  %I* : BOOL;		//TRUE when the voltage has fallen below the undervoltage threshold value from the CoE data
	CopperOn										AT  %I* : BOOL;		//TRUE when the external resistor is active, i.e. electrical energy is being converted to thermal energy in the resistor
	InputCycleCounter								AT  %I* : USINT;
	DCLinkVoltage									AT  %I* : UDINT;	//External supply voltage in mV
	ResistorCurrent									AT  %I* : DINT;		//Current through the external resistor in mA
	DutyCycle										AT  %I* : USINT;	//Temporal utilization of the external resistor in the last 100 ms in %
	I2TLoadFactor									AT  %I* : USINT;	

	WcState											AT  %I* : BOOL;
	InputToggle										AT  %I* : BOOL;
	state											AT  %I* : UINT;
	
END_VAR
VAR
{attribute 'hide'}
END_VAR

(* Ax_BrakeCopperIO						*)
(****************************************)
	
(* Work objects ****************************************)
	;
(*******************************************************)

END_FUNCTION_BLOCK

// POUs/IO/EL-EP/Eyx9xx
{attribute 'no_check'}
(* TwinSAFE terminal base IOs *)
FUNCTION_BLOCK Eyx9xx EXTENDS EcSlaveInfoDataExt //Safety logic device IO's
VAR_OUTPUT CONSTANT
	LOGIC_STATE_OFFLINE										: USINT := 0;
	LOGIC_STATE_RUN											: USINT := 1;
	LOGIC_STATE_STOP										: USINT := 2;
	LOGIC_STATE_SAFE										: USINT := 3;
	LOGIC_STATE_ERROR										: USINT := 4;
	LOGIC_STATE_START										: USINT := 6;
	LOGIC_STATE_PREPARE										: USINT := 8;
	LOGIC_STATE_RESTORE										: USINT := 11;
	LOGIC_STATE_CRC_OK										: USINT := 11;	
END_VAR
VAR_INPUT
END_VAR                         					
VAR_OUTPUT                      					
(* Device Info Data. Only available if the checkbox under the register TwinSafe_Logic is selected *)
{attribute 'displaymode':='hex'}
	ProjectCRC 										AT  %I* : WORD;		// Device Info Data
	SerialNumber									AT  %I* : UDINT;	// Device Info Data
                                					
(* standard DEVICE Inputs *)    					
	SafeLogicState									AT  %I* : USINT; 	//FSLOGIC Inputs
	CycleCounter									AT  %I* : USINT;	//FSLOGIC Inputs			
END_VAR
VAR
END_VAR

Super^(); //Get device name

{attribute 'monitoring' := 'call'}
PROPERTY PUBLIC inStateCrcOK : Bool
GET
inStateCrcOK :=	SafeLogicState = LOGIC_STATE_CRC_OK;
END_GET
END_PROPERTY

{attribute 'monitoring' := 'call'}
PROPERTY PUBLIC inStateError : Bool
GET
inStateError :=	SafeLogicState = LOGIC_STATE_ERROR;
END_GET
END_PROPERTY

{attribute 'monitoring' := 'call'}
PROPERTY PUBLIC inStateOffline : BOOL
GET
inStateOffline :=	SafeLogicState = LOGIC_STATE_OFFLINE;
END_GET
END_PROPERTY

{attribute 'monitoring' := 'call'}
PROPERTY PUBLIC inStatePrepare : Bool
GET
inStatePrepare :=	SafeLogicState = LOGIC_STATE_PREPARE;
END_GET
END_PROPERTY

{attribute 'monitoring' := 'call'}
PROPERTY PUBLIC inStateRestore : Bool
GET
inStateRestore :=	SafeLogicState = LOGIC_STATE_STOP;
END_GET
END_PROPERTY

{attribute 'monitoring' := 'call'}
PROPERTY PUBLIC inStateRun : BOOL
GET
inStateRun :=	SafeLogicState = LOGIC_STATE_RUN;
END_GET
END_PROPERTY

{attribute 'monitoring' := 'call'}
PROPERTY PUBLIC inStateSafe : Bool
GET
inStateSafe :=	SafeLogicState = LOGIC_STATE_SAFE;
END_GET
END_PROPERTY

{attribute 'monitoring' := 'call'}
PROPERTY PUBLIC inStateStart : Bool
GET
inStateStart :=	SafeLogicState = LOGIC_STATE_START;
END_GET
END_PROPERTY

{attribute 'monitoring' := 'call'}
PROPERTY PUBLIC inStateStop : Bool
GET
inStateStop :=	SafeLogicState = LOGIC_STATE_STOP;
END_GET
END_PROPERTY

END_FUNCTION_BLOCK

// POUs/IO/EL-EP/ZB8610
{attribute 'no_check'}
//ZB8610 - Fan cartridge for EtherCAT and Bus Terminals
//This function block controls the Beckhoff cartridge fan
FUNCTION_BLOCK ZB8610
VAR_INPUT
	Mode				: INT := MODE_TEMP;
END_VAR
VAR_OUTPUT
	Diag		AT%I*	: BOOL;	// [FALSE = Error | TRUE = Operational]	
END_VAR
VAR_OUTPUT CONSTANT
	MODE_TEMP			: INT := 0;
	MODE_1HZ			: INT := 1;
	MODE_2HZ			: INT := 2;
	MODE_3HZ			: INT := 3;
	MODE_4HZ			: INT := 4;
	MODE_5HZ			: INT := 5;
	MODE_6HZ			: INT := 6;
	MODE_7HZ			: INT := 7;
	MODE_8HZ			: INT := 8;
	MODE_9HZ			: INT := 9;
	MODE_HIGH			: INT := 10;
END_VAR
VAR
	Out			AT%Q*	: BOOL;
	Timer				: TON;
	CycleTime			: TIME;
	InstGETCURTASKINDEX	: GETCURTASKINDEX;
END_VAR

IF InstGETCURTASKINDEX.index = 0 THEN 
	InstGETCURTASKINDEX(index => ); 
	CycleTime			:= TO_TIME(TO_REAL(TwinCAT_SystemInfoVarList._TaskInfo[InstGETCURTASKINDEX.index].CycleTime) * 0.0001);
	CycleTime			:= CycleTime * 2;
END_IF	

CASE Mode OF
	MODE_TEMP			:	Timer(IN := FALSE, 			PT := T#0MS);
	MODE_1HZ			: 	Timer(IN := NOT Timer.Q, 	PT := T#500MS 	- CycleTime);
	MODE_2HZ			: 	Timer(IN := NOT Timer.Q, 	PT := T#250MS 	- CycleTime);
	MODE_3HZ			: 	Timer(IN := NOT Timer.Q, 	PT := T#166MS 	- CycleTime);
	MODE_4HZ			: 	Timer(IN := NOT Timer.Q, 	PT := T#125MS 	- CycleTime);
	MODE_5HZ			: 	Timer(IN := NOT Timer.Q, 	PT := T#100MS	- CycleTime);
	MODE_6HZ			: 	Timer(IN := NOT Timer.Q, 	PT := T#83MS 	- CycleTime);
	MODE_7HZ			: 	Timer(IN := NOT Timer.Q, 	PT := T#71MS 	- CycleTime);
	MODE_8HZ			: 	Timer(IN := NOT Timer.Q, 	PT := T#62MS 	- CycleTime);
	MODE_9HZ			: 	Timer(IN := NOT Timer.Q, 	PT := T#55MS 	- CycleTime);
	MODE_HIGH			: 	;
END_CASE
Out 					:= SEL(Timer.Q, Out, NOT Out) OR Mode = MODE_HIGH;

{attribute 'monitoring' := 'call'}
PROPERTY PUBLIC mode1Hz : BOOL
GET
Mode1Hz := Mode = MODE_1HZ;
END_GET
SET
Mode := SEL(Mode1Hz,MODE_TEMP ,MODE_1HZ);
END_SET
END_PROPERTY

{attribute 'monitoring' := 'call'}
PROPERTY PUBLIC mode2Hz : BOOL
GET
Mode3Hz := Mode = MODE_3HZ;
END_GET
SET
Mode := SEL(Mode2Hz,MODE_TEMP ,MODE_2HZ);
END_SET
END_PROPERTY

{attribute 'monitoring' := 'call'}
PROPERTY PUBLIC mode3Hz : BOOL
GET
Mode3Hz := Mode = MODE_3HZ;
END_GET
SET
Mode := SEL(Mode3Hz,MODE_TEMP ,MODE_3HZ);
END_SET
END_PROPERTY

{attribute 'monitoring' := 'call'}
PROPERTY PUBLIC mode4Hz : BOOL
GET
Mode4Hz := Mode = MODE_4HZ;
END_GET
SET
Mode := SEL(Mode4Hz,MODE_TEMP ,MODE_4HZ);
END_SET
END_PROPERTY

{attribute 'monitoring' := 'call'}
PROPERTY PUBLIC mode5Hz : BOOL
GET
Mode5Hz := Mode = MODE_5HZ;
END_GET
SET
Mode := SEL(Mode5Hz,MODE_TEMP ,MODE_5HZ);
END_SET
END_PROPERTY

{attribute 'monitoring' := 'call'}
PROPERTY PUBLIC mode6Hz : BOOL
GET
Mode6Hz := Mode = MODE_6HZ;
END_GET
SET
Mode := SEL(Mode6Hz,MODE_TEMP ,MODE_6HZ);
END_SET
END_PROPERTY

{attribute 'monitoring' := 'call'}
PROPERTY PUBLIC mode7Hz : BOOL
GET
Mode7Hz := Mode = MODE_7HZ;
END_GET
SET
Mode := SEL(Mode7Hz,MODE_TEMP ,MODE_7HZ);
END_SET
END_PROPERTY

{attribute 'monitoring' := 'call'}
PROPERTY PUBLIC mode8Hz : BOOL
GET
Mode8Hz := Mode = MODE_8HZ;
END_GET
SET
Mode := SEL(Mode8Hz,MODE_TEMP ,MODE_8HZ);
END_SET
END_PROPERTY

{attribute 'monitoring' := 'call'}
PROPERTY PUBLIC mode9Hz : BOOL
GET
Mode9Hz := Mode = MODE_9HZ;
END_GET
SET
Mode := SEL(Mode9Hz,MODE_TEMP ,MODE_9HZ);
END_SET
END_PROPERTY

{attribute 'monitoring' := 'call'}
PROPERTY PUBLIC modeHigh : BOOL
GET
ModeHigh := Mode = MODE_HIGH;
END_GET
SET
Mode := SEL(ModeHigh,MODE_TEMP ,MODE_HIGH);
END_SET
END_PROPERTY

{attribute 'monitoring' := 'call'}
PROPERTY PUBLIC modeTemp : BOOL //Default - Out = 0
GET
ModeHigh := Mode = MODE_TEMP;
END_GET
SET
Mode := MODE_TEMP;
END_SET
END_PROPERTY

END_FUNCTION_BLOCK

// POUs/IO/FreqConv/EtherCAT/DS402/EcFcDS402_ComBase
FUNCTION_BLOCK EcFcDS402_ComBase	EXTENDS EcSlaveInfoData IMPLEMENTS I_ActuatorEnableDisable(* SEW *)
VAR_INPUT
	ResetTrig												:	BOOL := TRUE;	//Resets error with rising edge 
	Enable													:	BOOL := FALSE;	//enables drive
	Start													:	BOOL := FALSE;	//motor rotates in right direction when TRUE
	StartBwd												:	BOOL := FALSE; 	//motor rotates in left direction when TRUE
	Feed													:	BOOL := TRUE;	//enables feed in right direction and should be set to FALSE when right limit sensor is reached
	FeedBwd													:	BOOL := TRUE;	//enables feed in left direction and should be set to FALSE when left limit sensor is reached
	Velo													: 	LREAL := 0.0;  	//sets speed of rotation
	ProtSwitchOK											: 	FUSE;			//monitors feeding protective device
	FuseBreakOK												: 	FUSE;			//monitors feeding circuit breaker 
	Contactor												:	BOOL := FALSE;	//if available
END_VAR
VAR_OUTPUT		
	{attribute 'displaymode':='binary'}
	Status													:	BYTE; (* for HMI *)
	Fault													:	BOOL; (* Drive Error *)
	SwitchedOn												:	BOOL; (* Drive enabled *)
	Ready													:	BOOL; (* Drive Ready *)
	Busy													:	BOOL;
	Error													:	BOOL;
	{attribute 'displaymode':='binary'}    
	Controlword										AT %Q* 	:	UINT; //Link to FC contro word
	{attribute 'displaymode':='binary'}																					
	Statusword										AT %I* 	:	UINT; //Link to FC status word 		
	Q_Contactor 									AT  %Q* :	BOOL; //Hardware output contactor 
    
END_VAR
VAR	
	ResetIntern												:	BOOL;
														
END_VAR
VAR_OUTPUT CONSTANT
END_VAR

METHOD PUBLIC reset : booL
VAR_INPUT
END_VAR
ProtSwitchOK.reset();
FuseBreakOK.reset();
ResetIntern												:= TRUE;
reset													:= TRUE;
END_METHOD

METHOD PUBLIC setContactorOFF : BOOL //Return true if contactor is off and not busy
VAR_INPUT
END_VAR
Q_Contactor := Contactor 									:=FALSE;				
SetContactorOFF 											:= switchOff() AND setDisable();
END_METHOD

METHOD PUBLIC setContactorON : bool //return true if contactor on
VAR_INPUT
END_VAR
Q_Contactor := Contactor 									:= ProtSwitchOK.Q AND FuseBreakOK.Q ;
SetContactorON												:= Q_Contactor;
END_METHOD

METHOD public setDisable : BOOL
VAR_INPUT
END_VAR
Enable										:= FALSE;
setDisable									:= TRUE;
END_METHOD

METHOD public setEnable : BOOL
VAR_INPUT
END_VAR
Enable										:= Q_Contactor;
setEnable									:= Enable;
END_METHOD

METHOD PUBLIC switchOff : BOOL //Return true if stopped / busy = false
VAR_INPUT
END_VAR
Start 														:= FALSE;
StartBwd													:= FALSE;
switchOff													:= NOT Busy;
END_METHOD

METHOD PUBLIC switchOn : BOOL
VAR_INPUT
END_VAR
switchOn := FALSE;
END_METHOD

{attribute 'monitoring' := 'call'}
PROPERTY public inError : bool
GET
inError := Error or not ProtSwitchOK.Q or not FuseBreakOK.Q;
END_GET
END_PROPERTY

{attribute 'monitoring' := 'call'}
PROPERTY public isBusy : bool
GET
isBusy := Busy;
END_GET
END_PROPERTY

{attribute 'monitoring' := 'call'}
PROPERTY public isDisabled : BOOL
GET
isDisabled := not Enable;
END_GET
END_PROPERTY

{attribute 'monitoring' := 'call'}
PROPERTY public isEnabled : BOOL
GET
isEnabled := Enable;
END_GET
END_PROPERTY

{attribute 'monitoring' := 'call'}
PROPERTY public isOff : BOOL
GET
isOff := TRUE;
END_GET
END_PROPERTY

{attribute 'monitoring' := 'call'}
PROPERTY public isOn : BOOL
GET
isOn := isEnabled;
END_GET
END_PROPERTY

{attribute 'monitoring' := 'call'}
PROPERTY noFeed : BOOL
GET
noFeed := not Feed and not FeedBwd;
END_GET
END_PROPERTY

{attribute 'monitoring' := 'call'}
PROPERTY ok : bool
GET
ok := isBusy;
END_GET
END_PROPERTY

END_FUNCTION_BLOCK

// POUs/IO/Fuse
{attribute 'no_check'}
//Fuse/Circuit breaker 
FUNCTION_BLOCK Fuse
VAR_INPUT
	Force													:	BOOL := FALSE;	//simulates Input
	Invert													:	BOOL := FALSE; 	//inverts the Hardware Input
	ResetTrig												:	BOOL := TRUE;	//Resets error with rising edge 
END_VAR     								
VAR_OUTPUT  								
	Q														:	BOOL;			//output
	Event													:	BOOL;			//TRUE when state is abnormal and error is not reset 
	In											AT  %I* 	: 	BOOL := TRUE;	//Hardware Input
END_VAR     								
VAR
END_VAR

(* signallocked Input-FB (MSS,Sicherung)				*)
(********************************************************)

(************************************)
IF NOT (In OR Force) XOR Invert
THEN
	Event													:= TRUE;
	Q														:= Invert;
ELSIF Event                         						
THEN                                						
	Event 													:= NOT ResetTrig;
ELSE                                						
	Q														:= Not Invert;
END_IF

(************************************)

METHOD PUBLIC reset : BOOL
VAR_INPUT
END_VAR
Event := FALSE;
reset := TRUE;
END_METHOD

END_FUNCTION_BLOCK

// POUs/IO/FreqConv/IOFcCom
{attribute 'no_check'}
FUNCTION_BLOCK IOFcCom IMPLEMENTS I_ActuatorFwdRev (* Frequence Converter IO Com *)
VAR_INPUT
	ResetTrig												:	BOOL := TRUE;		//Resets error with rising edge 
	Start													:	BOOL ;				//motor rotates in left direction when TRUE
	StartRev												:	BOOL ;				//motor rotates in right direction when TRUE
	Feed													:	BOOL := TRUE;		//enables feed in right direction and should be set to FALSE when right limit sensor is reached
	FeedBwd													:	BOOL := TRUE;		//enables feed in left direction and should be set to FALSE when left limit sensor is reached
	Velo													:	LREAL := 0.0;		//sets velocity of drive
	VeloMin													:	LREAL := 0.0;		//sets minimum limit of velocity of drive
	VeloMax													:	LREAL := 100.0;		//sets maximum limit of velocity of drive
	Contactor												:	BOOL;				//if available
	PT_DelBreak												:	TIME := T#1000MS;	//delay time before switching off 
	PT_DelEnable											:	TIME := T#1000MS;	//delay time for enabling
	ProtSwitchOK											: 	FUSE;				//monitors feeding protective device
	FuseBreakOK												: 	FUSE;				//monitors feeding circuit breaker 
END_VAR         								
VAR_OUTPUT      								
{attribute 'displaymode':='binary'}
	Status													:	BYTE;				//for HMI
	Ready											AT  %I* : 	BOOL := TRUE;		//TRUE when drive is ready to operate
	Busy													:	BOOL;				//Busy is TRUE at the rising edge of Enable and stays TRUE as long as the FB is performing any action. 
	Error											AT  %I* : 	BOOL := FALSE;		//Error identification 
END_VAR
VAR (* IO Internal *)
	Q_SetValue										AT  %Q* : 	INT;
	Q_Reset											AT  %Q* :	BOOL;
	Q_Enable										AT  %Q* :	BOOL;
	Q_Reverse										AT  %Q* :	BOOL;
	Q_Forward										AT  %Q* :	BOOL;
	Q_Break											AT  %Q* :	BOOL; 				//if available
	Q_Contactor										AT  %Q* :	BOOL;
END_VAR             								
VAR                 								
	TOF_Break												:	TOF;
	TOF_Enable												:	TOF;
	QuitIntern												:	BOOL;
	BreakOpenIntern											:	BOOL;
END_VAR

(* Com FC IO 										 		V1.3	*)
(********************************************************************)

(* Protection Switch ************************************************)
	IF ResetTrig 
	THEN 
		reset(); 
	END_IF

	ProtSwitchOK();
		
	FuseBreakOK(); (* same parameter like ProtSwitch *)

(* Contactor ********************************************************)
	Q_Contactor 											:= Contactor AND ProtSwitchOK.Q AND FuseBreakOK.Q;
	
(* Start ********************************************)
	IF 	StartRev 
		AND NOT Start
	THEN
		startForward();
	ELSIF Start 
		AND NOT StartRev
	THEN
		startReverse();
	ELSE
		 switchOff();
   END_IF

(* Enable ****************************************************)
	TOF_Enable(	
		IN := Q_SetValue <> 0,
		PT := PT_DelEnable);

	Q_Enable 												:= TOF_Enable.Q AND Ready AND Q_Break;

(* setvalue standardization *********************************)
	IF VeloMax > VeloMin THEN
		IF Velo >= VeloMax THEN
			Q_SetValue 										:= 32767;
		ELSIF Velo < VeloMin                				
		THEN                                				
			Q_SetValue 										:= 0;
		ELSE                                				
			Q_SetValue										:=LREAL_TO_INT ((32767.0 / (VeloMax - VeloMin)) * (Velo - VeloMin));
		END_IF                              				
	ELSE                                    				
		Q_SetValue 											:= 0;
	END_IF                                  				

(* setvalue **************************************)
	IF Q_Reverse THEN
		Q_SetValue 											:= ABS(Q_SetValue) * -1;
	ELSIF Q_Forward THEN              			
		Q_SetValue 											:= ABS(Q_SetValue);
	ELSE                                			
		Q_SetValue 											:= 0;
	END_IF                              	

(* HmiStatus **************************************************)
	Status.0 												:= Q_Reverse AND Ready AND Q_Contactor;
	Status.1 												:= Q_Forward AND Ready AND Q_Contactor;
	Status.2 												:= FALSE;
	Status.3 												:= Q_Break;
	Status.4 												:= FeedBwd ;
	Status.5 												:= Feed;
	Status.6 												:= Ready;
	Status.7 												:= Error;
	                                				
(* Status ***********************************************************)
	Busy 													:= TOF_Enable.Q AND TOF_Break.ET <= MAX(T#500MS,TOF_Break.PT) - T#500MS ;
	
(* Break ************************************************************)
	TOF_Break(	
		IN := Q_SetValue <> 0,
		PT := PT_DelBreak);

	IF Q_SetValue <> 0 
	THEN 
		BreakOpenIntern 									:= FALSE; 
	END_IF

	Q_Break 												:= TOF_Break.Q AND Ready OR BreakOpenIntern;

(* Reset ***********************************************************)
	Q_Reset 												:= ResetTrig OR QuitIntern;
	QuitIntern 												:= FALSE;

(**************************************************************)

METHOD PUBLIC closeBreak : booL //return true if brake open output is off
VAR_INPUT
END_VAR
BreakOpenIntern 											:= FALSE;
closeBreak													:= NOT Q_Break;
END_METHOD

METHOD PUBLIC openBreak : bool //Return true if break open is on
VAR_INPUT
END_VAR
BreakOpenIntern 							:= TRUE;
openBreak									:= Q_Break;
END_METHOD

METHOD PUBLIC reset : bool
VAR_INPUT
END_VAR
Error									:= FALSE;
reset							:= ProtSwitchOK.reset() and FuseBreakOK.reset();
END_METHOD

METHOD PUBLIC setContactorOFF : BOOL //Return true if contactor is off and not busy
VAR_INPUT
END_VAR
Contactor 													:= FALSE;
SetContactorOFF 											:= Not Q_Contactor and not busy;
END_METHOD

METHOD PUBLIC setContactorON : bool //return true if contactor on
VAR_INPUT
END_VAR
Contactor 													:= TRUE;
SetContactorON												:= Q_Contactor;
END_METHOD

METHOD PUBLIC startForward : bool //Return busy flag
VAR_INPUT
END_VAR
Start 														:= TRUE; 
StartRev := Q_Reverse										:= FALSE;
Q_Forward 													:= Q_Contactor AND Ready AND NOT inError AND Feed;
Busy														:= Q_Forward;
startForward												:= Busy;
END_METHOD

METHOD PUBLIC startReverse : bool //Return busy flag
VAR_INPUT
END_VAR
StartRev 													:= TRUE; 
Start := Q_Forward											:= FALSE;
Q_Reverse 													:= Q_Contactor AND Ready AND NOT inError AND Feed;
Busy														:= Q_Reverse;
startReverse												:= Busy;
END_METHOD

METHOD PUBLIC switchOff : BOOL //Return true if stopped / busy = false
VAR_INPUT
END_VAR
Start := StartRev											:= FALSE;
Q_Contactor := Q_Reverse := Q_Forward 						:= FALSE;
Busy														:= FALSE;
switchOff													:= TRUE;
END_METHOD

METHOD PUBLIC switchOn : BOOL  //True if motor is switched on
VAR_INPUT
END_VAR
switchOn := startForward();
END_METHOD

{attribute 'monitoring' := 'call'}
PROPERTY public forwardStarted : BOOL
GET
forwardStarted := Q_Contactor and Q_Forward;
END_GET
END_PROPERTY

{attribute 'monitoring' := 'call'}
PROPERTY public inError : bool
GET
inError := Error or not ProtSwitchOK.Q or not FuseBreakOK.Q;
END_GET
END_PROPERTY

{attribute 'monitoring' := 'call'}
PROPERTY public isBusy : bool
GET
isBusy := Busy;
END_GET
END_PROPERTY

{attribute 'monitoring' := 'call'}
PROPERTY public isOff : BOOL
GET
isOff := NOT Q_Contactor AND NOT Q_Reverse	and not Q_Forward;
END_GET
END_PROPERTY

{attribute 'monitoring' := 'call'}
PROPERTY public isOn : BOOL
GET
isOn := Q_Contactor and(Q_Forward or Q_Reverse);
END_GET
END_PROPERTY

{attribute 'monitoring' := 'call'}
PROPERTY noFeed : BOOL
GET
noFeed := NOT Feed and not FeedBwd;
END_GET
END_PROPERTY

{attribute 'monitoring' := 'call'}
PROPERTY ok : bool
GET
ok := isBusy;
END_GET
END_PROPERTY

{attribute 'monitoring' := 'call'}
PROPERTY public reverseStarted : BOOL
GET
reverseStarted := Q_Contactor and Q_Reverse;
END_GET
END_PROPERTY

END_FUNCTION_BLOCK

// POUs/IO/Motors/IOMotor
{attribute 'no_check'}
FUNCTION_BLOCK IOMotor IMPLEMENTS I_ActuatorOnOff
VAR_INPUT
	ResetTrig												:	BOOL := TRUE; //Confirm error
	start													:	BOOL;
	Feed													:	BOOL;
	ProtSwitchOK											: 	FUSE;
END_VAR                 							
VAR_OUTPUT
{attribute 'displaymode':='binary'}
	Status													:	BYTE;              							
	Q_Contactor										AT  %Q* :	BOOL; //Hardware output for main contactor to start motor	
	Busy													:	BOOL;
	Error													:	BOOL;
END_VAR                 							
VAR (* IO Internal *)   							

                        	
END_VAR                 	
VAR                     	
END_VAR

(* Com Motor IO 					 		V2.2		*)
(********************************************************)

(* Protection Switch *****************************************)
	IF ResetTrig THEN reset(); END_IF

	ProtSwitchOK();

(* Enable ****************************************************)
	IF Start THEN
		switchOn();
	ELSE
		switchOff();
	END_IF
	
(* HMI status *********************************************)
	_writeStatus();
	
(********************************************************)

METHOD PROTECTED _writeStatus : BOOL
VAR_INPUT
END_VAR
	
(* HmiStatus **************************************************)
	Status.0												:= NOT Q_Contactor;
	Status.1												:= Q_Contactor;
	Status.2												:= FALSE;
	Status.3												:= FALSE;
	Status.4												:= FALSE;
	Status.5												:= Feed ;
	Status.6												:= NOT Error;
	Status.7												:= Error;

	(* Result *)
	_writeStatus											:= TRUE;
    												
(**************************************************************)
END_METHOD

METHOD enable : BOOL //Result value = successful execution of desired action 
VAR_INPUT
	IN							:	BOOL; //TRUE = Enable Pos/FWD/Up/Open/Left/Work FALSE = Opposite
END_VAR
IF in
THEN
	enable := switchOn();
ELSE
	enable := switchOff();
END_IF
END_METHOD

METHOD PUBLIC reset : bool
VAR_INPUT
END_VAR
Error									:= FALSE;
reset									:= ProtSwitchOK.reset();
END_METHOD

METHOD public switchOff : BOOL  //True if motor is switched off
VAR_INPUT
END_VAR
Start														:= FALSE;
Q_Contactor 												:= FALSE;
Busy														:= FALSE;
Error														:= NOT ProtSwitchOK.Q;
switchOff													:= TRUE;
END_METHOD

METHOD public switchOn : BOOL  //True if motor is switched on
VAR_INPUT
END_VAR
Start														:= TRUE;
Q_Contactor		 											:= ProtSwitchOK.Q AND Feed;
switchOn													:= Q_Contactor;
Busy														:= switchOn;
Error														:= NOT ProtSwitchOK.Q;
END_METHOD

{attribute 'monitoring' := 'call'}
PROPERTY public inError : bool
GET
inError := Error;
END_GET
END_PROPERTY

{attribute 'monitoring' := 'call'}
PROPERTY public isBusy : bool
GET
isBusy := Busy;
END_GET
END_PROPERTY

{attribute 'monitoring' := 'call'}
PROPERTY public isOff : BOOL
GET
isOff := not Q_Contactor;
END_GET
END_PROPERTY

{attribute 'monitoring' := 'call'}
PROPERTY public isOn : BOOL
GET
isOn := Q_Contactor;
END_GET
END_PROPERTY

{attribute 'monitoring' := 'call'}
PROPERTY noFeed : BOOL
GET
noFeed := NOT Feed;
END_GET
END_PROPERTY

{attribute 'monitoring' := 'call'}
PROPERTY ok : bool
GET
ok := isBusy;
END_GET
END_PROPERTY

END_FUNCTION_BLOCK

// POUs/IO/Motors/IOMotor2Dir
{attribute 'no_check'}
FUNCTION_BLOCK IOMotor2Dir EXTENDS IOMotor IMPLEMENTS I_ActuatorFwdRev
VAR_INPUT
	StartBwd													:	BOOL; 
	FeedBwd														:	BOOL := TRUE;
END_VAR                 					
VAR_OUTPUT              					
	Q_ContactorBwd									AT  %Q* 	:	BOOL; //Hardware output for contactor to move backwards
END_VAR                 					
VAR 					
END_VAR                 	
VAR                     	
END_VAR

(* Com Motor IO 2 Directions		 		V2.2 	*)
(****************************************************)

(* Protection Switch *****************************************)
	IF ResetTrig 
	THEN 
		reset(); 
	END_IF
	
	ProtSwitchOK();
	
(* Enable ****************************************************)
	IF 	Start 
		AND NOT StartBwd 
	THEN
		startForward();
	ELSIF StartBwd 
		AND NOT Start 
	THEN
		startReverse();
	ELSE
		switchOff();
	END_IF
	
(* HMI status *********************************************)
	_writeStatus();
	
(********************************************************)

METHOD PROTECTED _writeStatus : BOOL
VAR_INPUT
END_VAR
	
(* HmiStatus **************************************************)
	Status.0 												:= Q_Contactor;
	Status.1 												:= Q_ContactorBwd;
	Status.2 												:= FALSE;
	Status.3 												:= FALSE;
	Status.4 												:= Feed;
	Status.5 												:= FeedBwd;
	Status.6 												:= NOT Error;
	Status.7 												:= Error;
	
	(* Result *)
	_writeStatus											:= TRUE;
    												
(**************************************************************)
END_METHOD

METHOD PUBLIC startForward : bool //Return busy flag
VAR_INPUT
END_VAR
Start														:= TRUE;
StartBwd  := Q_ContactorBwd									:= FALSE;
Q_Contactor													:= ProtSwitchOK.Q AND Feed;
startForward												:= Q_Contactor;
Busy														:= startForward;
Error														:= NOT ProtSwitchOK.Q;
END_METHOD

METHOD PUBLIC startReverse : bool //Return busy flag
VAR_INPUT
END_VAR
StartBwd 													:= TRUE;
Start  := Q_Contactor										:= FALSE;
Q_ContactorBwd 												:= ProtSwitchOK.Q AND FeedBwd;
startReverse												:= Q_ContactorBwd;
Busy														:= startReverse;
Error														:= NOT ProtSwitchOK.Q;
END_METHOD

METHOD PUBLIC switchOff : BOOL //Return true if stopped / busy = false
VAR_INPUT
END_VAR
Start := startBwd											:= FALSE;
Q_Contactor := Q_ContactorBwd 								:= FALSE;
Busy														:= FALSE;
switchOff													:= TRUE;
END_METHOD

METHOD PUBLIC switchOn : BOOL  //True if motor is switched on
VAR_INPUT
END_VAR
switchOn := startForward();
END_METHOD

{attribute 'monitoring' := 'call'}
PROPERTY public forwardStarted : BOOL
GET
forwardStarted := not Q_ContactorBwd and Q_Contactor;
END_GET
END_PROPERTY

{attribute 'monitoring' := 'call'}
PROPERTY public isOff : BOOL
GET
isOff := not Q_Contactor and not Q_ContactorBwd;
END_GET
END_PROPERTY

{attribute 'monitoring' := 'call'}
PROPERTY public isOn : BOOL
GET
isOn := Q_Contactor or Q_ContactorBwd;
END_GET
END_PROPERTY

{attribute 'monitoring' := 'call'}
PROPERTY noFeed : BOOL
GET
noFeed := NOT Feed and not FeedBwd;
END_GET
END_PROPERTY

{attribute 'monitoring' := 'call'}
PROPERTY public reverseStarted : BOOL
GET
reverseStarted := Q_ContactorBwd and not Q_Contactor;
END_GET
END_PROPERTY

END_FUNCTION_BLOCK

// POUs/IO/Motors/IOMotorStarDelta
{attribute 'no_check'}
FUNCTION_BLOCK IOMotorStarDelta EXTENDS IOMotor
VAR_INPUT
	PT_RestartDel											:	TIME := T#0S; //Delay to restart motor to avoid over heating
	PT_Delta												: 	TIME := T#5S; 
	ProtSwitchOK2											: 	FUSE;
END_VAR                 						
VAR_OUTPUT              						
	Q_StarContactor									AT %Q* 	: 	BOOL;
	Q_DeltaContactor								AT %Q* 	: 	BOOL;
	RestartDelActive										:	BOOL;
	ET_RestartDel											: 	TIME;	(* waiting-time of start interlock *)
END_VAR                 						
VAR                     						
	TON_StarDelta											:	TON;
	TP_RestartDel											:	TP;
END_VAR

(* Start Delta Motor IO	 				 	V1.1	*)
(****************************************************)

(* Protection Switch *****************************************)
	IF ResetTrig  THEN reset(); END_IF

	ProtSwitchOK();
	ProtSwitchOK2();
	
(* Start ****************************************************)
	IF Start THEN
		switchOn();
                       										
		Q_StarContactor 									:= 	Q_Contactor
																AND NOT TON_StarDelta.Q
																AND NOT Q_DeltaContactor;

		Q_DeltaContactor 									:= 	Q_Contactor
																AND TON_StarDelta.Q;

		TP_RestartDel();
	ELSE
		switchOff();
	END_IF

(* Timer *****************************************************)
	TON_StarDelta(IN := Q_Contactor, PT := PT_Delta);

	//Restart delay
	TP_RestartDel(IN := TP_RestartDel.Q,PT := PT_RestartDel); //Execute restart delay
	RestartDelActive										:= TP_RestartDel.Q;
	
	IF TP_RestartDel.ET > T#0MS 
	THEN
		ET_RestartDel		:= TP_RestartDel.PT - TP_RestartDel.ET;
	ELSE
		ET_RestartDel		:= t#0ms;
	END_IF
	
(* HMI status *********************************************)
	_writeStatus();
	
(********************************************************)

METHOD PROTECTED _writeStatus : BOOL
VAR_INPUT
END_VAR
(* HmiStatus **************************************************)
	Status.0												 := NOT Q_Contactor;
	Status.1												 := Q_Contactor;
	Status.2												 := Q_DeltaContactor;
	Status.3												 := RestartDelActive;
	Status.4												 := FALSE;
	Status.5												 := Feed;
	Status.6												 := NOT Error AND NOT RestartDelActive;
	Status.7												 := Error;

	(* Result *)
	_writeStatus											:= TRUE;
    												
(**************************************************************)
END_METHOD

METHOD PUBLIC reset : booL
VAR_INPUT
END_VAR

reset									:= ProtSwitchOK.reset() AND ProtSwitchOK2.reset();
Error									:= FALSE;
END_METHOD

METHOD PUBLIC resetRestartTmr : booL
VAR_INPUT
END_VAR
MEMSET(ADR(TP_RestartDel),0,SIZEOF(TP_RestartDel));
resetRestartTmr										:= TRUE;
END_METHOD

METHOD public switchOff : BOOL
VAR_INPUT
END_VAR
Start														:= FALSE;
TP_RestartDel(IN := Q_Contactor , PT := PT_RestartDel);
Q_Contactor 												:= FALSE;
Q_StarContactor												:= FALSE;
Q_DeltaContactor											:= FALSE;
Busy														:= FALSE;
Error														:= NOT ProtSwitchOK.Q OR NOT ProtSwitchOK2.Q;
switchOff													:= TRUE;
END_METHOD

METHOD public switchOn : BOOL //True if motor is switched on
VAR_INPUT
END_VAR
Start														:= TRUE;
Q_Contactor		 											:= ProtSwitchOK.Q AND ProtSwitchOK2.Q AND Feed AND NOT TP_RestartDel.Q;
switchOn													:= Q_Contactor;
Busy														:= switchOn;
Error														:= NOT ProtSwitchOK.Q OR NOT ProtSwitchOK2.Q;
END_METHOD

{attribute 'monitoring' := 'call'}
PROPERTY public isOn : BOOL
GET
isOn := Q_Contactor;
END_GET
END_PROPERTY

{attribute 'monitoring' := 'call'}
PROPERTY ok : bool
GET
ok := Q_Contactor and Q_DeltaContactor ;
END_GET
END_PROPERTY

END_FUNCTION_BLOCK

// POUs/IO/AnalogIn32
{attribute 'no_check'}
FUNCTION_BLOCK AnalogIn32
VAR_INPUT
	MinValue												: 	LREAL 	:= 0.0;
	MaxValue												: 	LREAL 	:= 0.0;
	NoOfDigits												: 	INT 	(0..10)	:= 0; //number of decimal digits of scaled Q variable 
	OutOnError												:	LREAL 	:= 0.000000000000000001;
{attribute 'displaymode':='binary'}     	            	
	Options													:	BYTE  := 2#0000_0010; (* .0 = FALSE Scale value from 0 to e.g. 32767 / TRUE scale singed value e.g. -32768 <-> 32767 , see Options .1 and .2 for more scaling Options 
																						.1 = FALSE = 32 bit resolution / TRUE = value is based on 24 bit resolution e.g. -> -8388608.0 or 0.0 <-> 8388607.0 
																						.2 = Right adjust of 32/24 bit value -> value will be shifted by 8 bits (divided bv 256)   
																						.3 = TRUE = Enable extended range mode -> change scaling to +/-7812500 instead of r+/- 838860x *)
	Offset													:	LREAL := 0.0;
END_VAR                 									
VAR                                     	            	
{attribute 'displaymode':='binary'}     	            	
	Status										AT  %I*		:	WORD := 2#0100_0000_0000_0000;	//Terminal status word -> can also be linked with status byte 
END_VAR                                 	            	
VAR_OUTPUT                              	            	
	Q														:	LREAL;	//scaled result value
	In											AT  %I* 	: 	DINT; 	//Hardware Input 
                                        	
	(* Statusbist *)                    	
	Underrange 												:	BOOL ;//Bit 0
	Overrange												:	BOOL ;//Bit 1
	Limit_1													:	BYTE ;(* Bit 2-3 			0: not active
																							1: value is smaller than limit 
																							2: value is bigger than limit 
																							3: value is equal to limit  *)
	Limit_2													:	BYTE ;(* Bit 4-5 			0: not active
																							1: value is smaller than limit 
																							2: value is bigger than limit 
																							3: value is equal to limit  *)             											
	Error													:	BOOL ;//Bit 6
	SyncError												:	BOOL ;//Bit 13
	TxPDOState												:	BOOL ;//Bit 14 - TRUE if NOT Valid
END_VAR                                 	                         
VAR                                     	                         
	TxPDOTgl												:	BOOL ;
END_VAR

(* read 32bit analog value 																				    *)
(* resolution process image			e.g.				/ 0V = 0 / 10V = 2147483647 / -10V = - 2147483647 	*)
(* or directly with NoOfDigits																	250 -> 25.0°*)
(************************************************************************************************************)

(* evaluate statusword **************************************************************************************)
	Underrange 												:= Status.0;
	Overrange												:= Status.1;
	Limit_1.0												:= Status.2;
	Limit_1.1												:= Status.3;
	Limit_2.0												:= Status.4;
	Limit_2.1												:= Status.5;
	Error													:= Status.6 OR MinValue = MaxValue AND NoOfDigits = 0;
	SyncError												:= Status.13;
	TxPDOState												:= Status.14; //True if not valid
	TxPDOTgl												:= Status.15;
	
(* Scaling ******************************************************************)
	IF MaxValue <> MinValue 
	THEN
		IF Options.1 
		THEN //24 bit resolution
			IF NOT Options.3
			THEN
				Q 	 										:= Offset + Scale(SEL(Options.2 , In , In / 256.0 ) , SEL(Options.0, 0.0, -8388608.0), 8388607.0, MinValue , MaxValue);
			ELSE
		 		Q 	 										:= Offset + Scale(SEL(Options.2 , In , In / 256.0 ) , SEL(Options.0, 0.0, -7812500.0), 7812500.0, MinValue , MaxValue);
			END_IF
		ELSE //32 bit resolution 
			Q 	 											:= Offset + Scale(SEL(Options.2 , In , In / 256.0 ) , SEL(Options.0, 0.0, -2147483648.0), 2147483647.0, MinValue , MaxValue);		
		END_IF
		IF NoOfDigits > 0
		THEN
			Q												:= TO_FMLREAL(Q,NoOfDigits);
		END_IF
	
	ELSIF NoOfDigits > 0 (* Bsp PT100 *)
	THEN
		Q													:= Offset + TO_FMLREAL(In,NoOfDigits);
		
	ELSE  													
		Q 													:= 0.0;
	END_IF

	IF 	Error AND OutOnError <> 0.000000000000000001
	THEN
		Q													:= OutOnError;
	END_IF
(**********************************************************************************************************************)

PROPERTY optEnable24BitResolution : BOOL //In value is provided as 32bit value instead if 24bit
GET
optEnable24BitResolution := Options.1;
END_GET
SET
Options.1 := optEnable24BitResolution;
END_SET
END_PROPERTY

PROPERTY PUBLIC optEnableScaleExtRangeMode : bool
GET
optEnableScaleExtRangeMode := Options.3;
END_GET
SET
Options.3 := optEnableScaleExtRangeMode;
END_SET
END_PROPERTY

PROPERTY PUBLIC optEnableScaleSignedValue : bool
GET
optEnableScaleSignedValue := Options.0;
END_GET
SET
Options.0 := optEnableScaleSignedValue;
END_SET
END_PROPERTY

PROPERTY PUBLIC optShiftValueBy8Bits : BOOL
GET
optShiftValueBy8Bits := Options.2;
END_GET
SET
Options.2 := optShiftValueBy8Bits;
END_SET
END_PROPERTY

END_FUNCTION_BLOCK

// POUs/IO/AnalogInELMBase
// Based FB for analog input channels of ELM terminals incl. EtherCAT Slave Info Data 
//You can inherit your final implementation from this base "class"  
FUNCTION_BLOCK AnalogInELMBase EXTENDS EcSlaveInfoData
VAR_INPUT
	Enable													:	BOOL 	:= TRUE;
	MinValue												: 	LREAL 	:= 0.0;
	MaxValue												: 	LREAL 	:= 0.0;
	NoOfDigits												: 	INT 	(0..10)	:= 0; //number of decimal digits of scaled Q variable 
	OutOnError												:	LREAL 	:= 0.000000000000000001;
{attribute 'displaymode':='binary'}     	            	
	Options													:	BYTE  := 2#0000_0000;
END_VAR                 									
VAR                                     	            	
{attribute 'displaymode':='binary'}     	            	
	Status										AT  %I*		:	DWORD := 2#0100_0000_0000_0000;	//Terminal status (4 bytes) 
	
END_VAR                                 	            	
VAR_OUTPUT                              	            	                                       	
	(* Statusbist *)                    	
	NoOfSamples												:	USINT; //Byte 1
	Error													:	BOOL; //Byte2.0
	Underrange 												:	BOOL; //Byte2.1
	Overrange												:	BOOL ; //Byte2.2
	Diag													:	BOOL; //Byte2.4
	TxPDOState												:	BOOL; //Byte2.5
	InputCycleCounter										:	USINT; //Byte2.6/.7	
END_VAR                                 	
VAR                                     	
END_VAR

(* Base FB for ELM analog in terminals 																		*)
(************************************************************************************************************)

(* evaluate statusword **************************************************************************************)
	MEMCPY(ADR(NoOfSamples),ADR(Status),SIZEOF(NoOfSamples));
	Error													:= Enable AND (Status.8 OR MinValue = MaxValue AND NoOfDigits = 0);
	Underrange 												:= Status.9;
	Overrange												:= Status.10;
	
	Diag													:= Status.12;
	TxPDOState												:= Status.13; //True if not valid
	InputCycleCounter.0										:= Status.14;
	InputCycleCounter.1										:= Status.15;
	
(**********************************************************************************************************************)

END_FUNCTION_BLOCK

// POUs/IO/AnalogInELMSingleSampleDINT
// AnalogIn FB to read and scale a single DINT (24bit) sample input from ELMxxxx terminal
// Set bit 3 (Options.3) to true to enable scaling based on +/-7812500 instead of legacy range values +/-838860x
FUNCTION_BLOCK AnalogInELMSingleSampleDINT EXTENDS AnalogInELMBase
VAR_INPUT
	Offset													:	LREAL := 0.0;

END_VAR                 									
VAR                                     	            	
END_VAR                                 	            	
VAR_OUTPUT                              	            	                                       	
	Q														:	LREAL;	//scaled result value
	In											AT  %I* 	: 	DINT; 	//Hardware Input 
END_VAR                                 	
VAR                                   	
END_VAR

(* Read single DINT sample value from ELM terminal and scale to user units									*)
(************************************************************************************************************)

(* evaluate statusword **************************************************************************************)
	SUPER^();
	
(* Scaling ******************************************************************)
	IF MaxValue <> MinValue 
	THEN	
		IF NOT Options.3
		THEN
			Q 	 											:= Offset + Scale(TO_LREAL(In) , -8388608.0, 8388607.0, MinValue , MaxValue);
		ELSE
			Q 	 											:= Offset + Scale(TO_LREAL(In), -7812500.0, 7812500.0, MinValue , MaxValue);
		END_IF	
		IF NoOfDigits > 0
		THEN
			Q												:= TO_FMLREAL(Q,NoOfDigits);
		END_IF
	
	ELSIF NoOfDigits > 0 (* Bsp PT100 *)
	THEN
		Q													:= Offset + TO_FMLREAL(In,NoOfDigits);
		
	ELSE  													
		Q 													:= 0.0;
	END_IF

	IF 	Error AND OutOnError <> 0.000000000000000001
	THEN
		Q													:= OutOnError;
	END_IF
(**********************************************************************************************************************)

METHOD FB_init : BOOL
VAR_INPUT
	bInitRetains : BOOL; // if TRUE, the retain variables are initialized (warm start / cold start)
	bInCopyCode : BOOL;  // if TRUE, the instance afterwards gets moved into the copy code (online change)
END_VAR
IF NOT bInCopyCode THEN
	NoOfDigits 							:= 2;
END_IF
END_METHOD

PROPERTY PUBLIC optEnableScaleExtRangeMode : bool
GET
optEnableScaleExtRangeMode := Options.3;
END_GET
SET
Options.3 := optEnableScaleExtRangeMode;
END_SET
END_PROPERTY

END_FUNCTION_BLOCK

// POUs/IO/AnalogInELMSingleSampleREAL
// AnalogIn FB to read and scale a single REAL sample input from ELMxxxx terminal
// Set bit 3 (Options.3) to true to enable scaling based on +/-7812500 instead of legacy range values +/-838860x
// NoOfDigits per default set to 3... 
FUNCTION_BLOCK AnalogInELMSingleSampleREAL EXTENDS AnalogInELMBase
VAR_INPUT
	Offset													:	LREAL := 0.0;
END_VAR                 									
VAR                                     	            	
END_VAR                                 	            	
VAR_OUTPUT                              	            	                                       	
	Q														:	LREAL;	//scaled result value
	In											AT  %I* 	: 	REAL; 	//Hardware Input 
END_VAR                                 	
VAR                                     	
END_VAR

(* Read single REAL sample value from ELM terminal and scale to user units									*)
(************************************************************************************************************)

(* evaluate statusword **************************************************************************************)
	SUPER^();
	
(* Scaling ******************************************************************)
	IF MaxValue <> MinValue 
	THEN			
		IF NOT Options.3
		THEN
			Q 	 											:= Offset + Scale(TO_LREAL(In), -8388608.0, 8388607.0, MinValue , MaxValue);
		ELSE
			Q 	 											:= Offset + Scale(TO_LREAL(In),  -7812500.0, 7812500.0, MinValue , MaxValue);		
		END_IF	
		
		IF NoOfDigits > 0
		THEN
			Q												:= TO_FMLREAL(Q,NoOfDigits);
		END_IF
	
	ELSIF NoOfDigits > 0 (* Bsp PT100 *)
	THEN
		Q													:= Offset + TO_FMLREAL(In,NoOfDigits);
		
	ELSE  													
		Q 													:= 0.0;
	END_IF


(**********************************************************************************************************************)

METHOD FB_init : BOOL
VAR_INPUT
	bInitRetains : BOOL; // if TRUE, the retain variables are initialized (warm start / cold start)
	bInCopyCode : BOOL;  // if TRUE, the instance afterwards gets moved into the copy code (online change)
END_VAR
IF NOT bInCopyCode THEN
	NoOfDigits 							:= 3;
END_IF
END_METHOD

PROPERTY PUBLIC optEnableScaleExtRangeMode : bool
GET
optEnableScaleExtRangeMode := Options.3;
END_GET
SET
Options.3 := optEnableScaleExtRangeMode;
END_SET
END_PROPERTY

END_FUNCTION_BLOCK

// POUs/IO/AnalogOut
{attribute 'no_check'}
//Provides an INT output varibale (Q	AT  %Q* : 	INT) to writed a scaled lreal value to an anallog output (terminal)
FUNCTION_BLOCK AnalogOut
VAR_INPUT
	SetValue												: 	LREAL 	:= 0.0;	
	MinValue												: 	LREAL 	:= 0.0;
	MaxValue												: 	LREAL 	:= 0.0;	
{attribute 'displaymode':='binary'}
	Options													:	BYTE 	:= 2#0000_0000; (* .0 = FALSE scale output to 0 - 32767 / TRUE = scale output from -32768 to +32767 *)
END_VAR             							
VAR_OUTPUT          							
	Q												AT  %Q* : 	INT; (* Hardware Output *)
END_VAR             							
VAR                 							
	x														:	LREAL;
END_VAR

(* Analogvalue output	 													    *)
(* resolution  							/ 0V = 0 / 10V = 32768 / -10V = - 32767 *)
(********************************************************************************)

(* standardization **************************************************************)
	Q															:= TO_INT(Scale(SetValue,MinValue,MAxValue,SEL(Options.0 , 0.0  , -32768.0), 32767.0));		

(*********************************************************************************)

PROPERTY PUBLIC optEnableScaleSignedValue : bool
GET
optEnableScaleSignedValue := Options.0;
END_GET
SET
Options.0 := optEnableScaleSignedValue;
END_SET
END_PROPERTY

END_FUNCTION_BLOCK

// POUs/IO/BlowOffSensors
{attribute 'no_check'}
//FB generates a pulse "Pulse" time based signal on every bit at Q (DWORD) for a certain lenght
//The sequecne will starts based on the seletcted time of interval if Enable is TRUE
//The FB can be used to activate air blow valves on by one to clean sensors in a dusty environment
FUNCTION_BLOCK BlowOffSensors
VAR_INPUT
	Enable													:	BOOL;			//FB will be processed as long as enable is TRUE
	StartManual												:	BOOL;			//starts FB without interval
	Interval												:	TIME := T#60M; 	//Blow of autostart interval
	Lenght													:	TIME := T#4S; 	//Duration of pulsing
	Pulse													:	TIME := T#500MS; //On/Off pulse duration
END_VAR                 									
VAR_OUTPUT              									
	Aktiv													:	BOOL;			//Busy is TRUE at the rising edge of Enable and stays TRUE as long as the FB is performing any action.  
{attribute 'displaymode':='binary'}    
	Q														:	DWORD := 0;		//Each bit will be set and reset based on the settings one by one 
END_VAR                 									
VAR                     									
	state													:	INT := 0;
	i														:	SINT ;
	TON_Interval											:	TON;
	TON_Lenght		 										: 	TON;
	TOF_Pulse	 											:	TOF;
END_VAR

(* Abblastaktgenerator					*)
(***************************************)

(* Intervalzeit ***********************************************************************)
IF Enable 
THEN
	CASE state OF
	0:
		TON_Interval(IN := FALSE);
		state 												:= 10;
		i 													:= -1;

	1:
		Aktiv := FALSE;
		TON_Interval(IN := Interval <> T#0MS , PT := Interval);
		IF TON_Interval.Q
			OR StartManual
		THEN
			TON_Interval(IN := FALSE);
			
			state 											:= 10;
			Aktiv 											:= TRUE;
			i 												:= -1;
		END_IF

	10:
		i := i + 1;
		IF i > 31 THEN
			state 											:= 1;
		ELSE
			TON_Lenght(IN := FALSE);
			TOF_Pulse(IN := FALSE);
			
			Q		 										:= 0;
			state 											:= 11;
		END_IF                  							

	11:
		TON_Lenght(IN := TRUE, PT := Lenght);

		IF 	TON_Lenght.Q
			AND Q = 0
		THEN
			state 											:= 10;
		ELSE
			IF 	NOT TOF_Pulse.Q 
				AND Q <> 0 
			THEN
				TOF_Pulse(IN:=TRUE  , PT:= Pulse);
				Q		 									:= 0;
			ELSIF NOT TOF_Pulse.Q 
				AND Q = 0 
			THEN
				TOF_Pulse(IN:= TRUE , PT:= Pulse) ;
				Q		 									:= SETBIT32(Q,i);
			END_IF
			(* Work Timer *)
			TOF_Pulse(IN:=FALSE);
		END_IF

	END_CASE
ELSE
	Aktiv 													:= FALSE;
	state 													:= 0;
	Q														:= 0;
END_IF

(**********************************************************************************************************)

END_FUNCTION_BLOCK

// POUs/TimeHelper/Pulse
{attribute 'no_check'}
//Generates a pulse signal 
FUNCTION_BLOCK Pulse
VAR_INPUT
	IN														: BOOL; //Start pulse generator
	PT_ON													: TIME; //Time pulse on	
	PT_OFF													: TIME; //Time pulse off 
END_VAR             										
VAR_OUTPUT          										
	Q														: BOOL; 
	RT														: BOOL; 
	FT														: BOOL;
END_VAR             										
VAR                 	
	TON_PULSE												: TON;
END_VAR

	(* Pulse generator																*)
	(********************************************************************************)

(* Reset flag *)
RT := FT													:= FALSE;
(* logic *)
IF 	Q AND(TON_PULSE.Q OR NOT IN)
THEN
	TON_PULSE(IN:=FALSE  , PT:= PT_OFF);
	FT 														:= Q;
	Q 														:= FALSE;
ELSIF NOT Q AND TON_PULSE.Q
	OR_ELSE In AND NOT TON_PULSE.IN 
THEN
	RT 														:= NOT Q;
	TON_PULSE(IN:= FALSE , PT:= PT_ON) ;
	Q 														:= TRUE;
END_IF

//Run timer
TON_PULSE(IN:=IN);

(***********************************************************************************************************************)

END_FUNCTION_BLOCK

// POUs/IO/Button
{attribute 'no_check'}
FUNCTION_BLOCK Button 
VAR_INPUT
	Enable													:	BOOL := TRUE;	//FB will be processed as long as enable is TRUE 
	RstTGL													:	BOOL := FALSE; 	//resets the Toggle signal
	SetTGL													:	BOOL := FALSE;	//sets the Toggle signal
	Force													:	BOOL := FALSE; 	//simulates Input signal
	Invert													:	BOOL := FALSE; 	//inverts the Hardware Input
	LED												AT  %Q*	:	BOOL;			//LED/Light hardware output
END_VAR         									
VAR_OUTPUT
	Q														:	BOOL;	//direct signal
	Q_RT													:	BOOL;	//R_Trig signal of delay Q
	Q_FT													:	BOOL;	//F_Trig signal of delay Q
	Q_TGL													:	BOOL;	//Toggle -> use flag Q_RT
	In												AT  %I*	:	BOOL; 	//Hardware Input
END_VAR
VAR
	Mem														:	BOOL;
END_VAR

(* Taster mit Togglefunktion V1.0						*)
(********************************************************)

(********************************************************)
Mem															:= Q;
Q 															:= ((In OR Force) XOR Invert) AND Enable;
Q_RT 														:= NOT Mem AND Q;
Q_FT														:= Mem AND NOT Q;
Q_TGL 														:= (Q_RT XOR Q_TGL);
(********************************************************)

METHOD PUBLIC setDisable : BOOL
VAR_INPUT
END_VAR
Enable 														:= FALSE;
setDisable													:= TRUE;
END_METHOD

METHOD PUBLIC setEnable : bool
VAR_INPUT
END_VAR
Enable 														:= TRUE;
setEnable													:= TRUE;
END_METHOD

METHOD PUBLIC setLedOFF : bool
VAR_INPUT
END_VAR
LED 														:= FALSE;
setLEDOff													:= TRUE;
END_METHOD

METHOD PUBLIC setLedON : booL
VAR_INPUT
END_VAR
LED 														:= TRUE;
setLedON													:= TRUE;
END_METHOD

METHOD PUBLIC TGL : booL //Return value = Q_TGL status
VAR_INPUT
END_VAR
TGL := Q_TGL 														:= NOT Q_TGL;
END_METHOD

METHOD PUBLIC TglOff : booL
VAR_INPUT
END_VAR
Q_TGL 														:= FALSE;
TglOFF														:= TRUE;
END_METHOD

METHOD PUBLIC TglOn : bool
VAR_INPUT
END_VAR
Q_TGL 														:= TRUE;
TglON														:= TRUE;
END_METHOD

END_FUNCTION_BLOCK

// POUs/IO/ButtonExt
{attribute 'no_check'}
//Button with delay function 
FUNCTION_BLOCK ButtonExt EXTENDS Button
VAR_INPUT
	PT_ON													:	TIME := T#0MS; 	//Delay for Q, Q_RT (TGL) and Q_FT
END_VAR
VAR_OUTPUT
	Q_DIRECT												:	BOOL; 	//Direct signal - undelayed
END_VAR
VAR
	TON														:	TON;
END_VAR

(* Button with toggle-function and on-delay		V1.5	*)
(********************************************************)

(********************************************************)
TON(IN := ((In OR Force) XOR Invert) AND Enable, PT := PT_ON);
Q_DIRECT 													:= TON.IN;
IF NOT Q    												
THEN        												
	Q 														:= TON.Q;
	Q_RT 													:= Q;
	Q_FT 													:= FALSE;
ELSE        												
	Q 														:= TON.IN;
	Q_RT 													:= FALSE;
	Q_FT 													:= NOT Q;
END_IF      	

Q_TGL := NOT RstTGL AND (Q_RT XOR Q_TGL OR SetTGL) ;

(********************************************************)

END_FUNCTION_BLOCK

// POUs/IO/InOut
{attribute 'no_check'}
FUNCTION_BLOCK InOut 
VAR_INPUT
	Q												AT  %Q*	:	BOOL; //Link to hardware output
END_VAR             								
VAR_OUTPUT          								
	In												AT  %I*	:	BOOL; //Link to hardware input
END_VAR
VAR
END_VAR

;

END_FUNCTION_BLOCK

// POUs/IO/InOutExt
{attribute 'no_check'}
FUNCTION_BLOCK InOutExt EXTENDS InOut IMPLEMENTS I_ActuatorOnOff
VAR_INPUT
	ResetTrig												:	BOOL;	//Resets error with rising edge
	Invert													:	BOOL ;			//Inverts the logic of varibale In (AT  %I*)
	PT_Timeout												:	TIME := T#3S;  	//Time value until Timeout of process (Error)
END_VAR                     				
VAR_OUTPUT                  				
	Busy													:	BOOL;			//Busy is TRUE at the rising edge of Execute and FALSE when one of the outputs Done, Aborted, or Error is set 
	ErrorOn													:	BOOL;			//Timeout error waiting for IN changing to TRUE
	ErrorOff												:	BOOL;			//Timeout error waiting for IN changing to FALSE
	Done													:	BOOL;			//The Done output is set when the commanded action has been completed successfully 
	Status													:	BYTE;			//8 different query Options (conditions see below)
END_VAR                     	
VAR                         	
	tonRM													:	ton;			
END_VAR

(* Actuator with feedback								*)
(********************************************************)

(********************************************************)
	IF Q 
	THEN
		SwitchOn();
	ELSE
		SwitchOff();
	END_IF
	_runtimeChk();
	_writeStatus();

(********************************************************)

METHOD PROTECTED _runtimeChk : BOOL
VAR_INPUT
END_VAR
	tonRM(
		IN	:= Busy AND NOT ResetTrig,  
		PT 	:= PT_Timeout,
		Q	=> );
		
	ErrorOff 												:= tonRM.Q AND NOT Q;
	ErrorOn 												:= tonRM.Q AND Q;

	_runtimeChk									:= TRUE;
END_METHOD

METHOD PROTECTED _writeStatus : BOOL
VAR_INPUT
END_VAR
	Status.0 												:= NOT Q;
	Status.1 												:= Q;
	Status.2 												:= NOT (In XOR Invert);
	Status.3 												:= In XOR Invert;
	Status.4 												:= NOT ErrorOff;
	Status.5 												:= NOT ErrorOn;
	Status.6 												:= NOT Status.7;
	Status.7 												:= ErrorOff OR ErrorOn;
	
	(* Result *)
	_writeStatus											:= TRUE;
END_METHOD

METHOD PUBLIC enable : BOOL //Result value = TRUE if successful executed (
VAR_INPUT 
	IN								: BOOL; //TRUE = ON/FALSE = OFF	
END_VAR
IF IN
THEN
	enable							:= switchOn();
ELSE
	enable							:= switchOff();
END_IF
END_METHOD

{attribute 'monitoring' := 'call'}
PROPERTY public inError : BOOL
GET
inError := ErrorON or ErrorOff;
END_GET
END_PROPERTY

{attribute 'monitoring' := 'call'}
PROPERTY public isBusy : bool
GET
isBusy := Busy;
END_GET
END_PROPERTY

{attribute 'monitoring' := 'call'}
PROPERTY public isOff : BOOL
GET
isOff := not Q;
END_GET
END_PROPERTY

{attribute 'monitoring' := 'call'}
PROPERTY public isOn : BOOL
GET
isOn := Q;
END_GET
END_PROPERTY

{attribute 'monitoring' := 'call'}
PROPERTY Public noFeed : BOOL
GET
noFeed := FALSE;
END_GET
END_PROPERTY

{attribute 'monitoring' := 'call'}
PROPERTY Public ok : bool
GET
ok := Q and Done or not Q and not Done;
END_GET
END_PROPERTY

METHOD PUBLIC reset : Bool
VAR_INPUT
END_VAR
tonRM(IN := FALSE);
reset := TRUE;
END_METHOD

METHOD public switchOff : BOOL
VAR_INPUT
END_VAR
	
	Q														:= FALSE;
	Done													:= NOT (In XOR Invert);
	Busy													:= NOT Done;
	switchOff												:= Done;
END_METHOD

METHOD public switchOn : BOOL
VAR_INPUT
END_VAR
	Q														:= TRUE;
	Done													:= (In XOR Invert);
	Busy													:= NOT Done;
	switchOn												:= Done;
END_METHOD

END_FUNCTION_BLOCK

// POUs/IpcDiag/MDP/InfoModuls/MDP_CPU
{attribute 'no_check'}
//Wrapper for available MDP_xxxx FBs of the lib, based on Beckhoff MDP - invalid values are reported via EventLogger 
//based on Tc2_MDP.lib - please see Beckhoff documentation for further information about Tc2_MDP.lib (IPC diagnostics)
FUNCTION_BLOCK MDP_CPU  EXTENDS FbBase
VAR_OUTPUT CONSTANT
	MIN_CPU													:	INT := 1;
	MAX_CPU													:	INT := 8;
END_VAR                 									
VAR_INPUT               									
	AmsNetId												: 	T_AmsNetId := '';				//AmsNetId as text
	Timeout													:	TIME := DEFAULT_ADS_TIMEOUT;	//Ads timeout
END_VAR                 									
VAR_OUTPUT              									
	Frequency												:  ARRAY[MIN_CPU..MAX_CPU] OF	UDINT;	//current CPU frequency
	Usage													:	ARRAY[MIN_CPU..MAX_CPU] OF	UINT;	//current CPU usage in %
	Temperature												:	ARRAY[MIN_CPU..MAX_CPU] OF	INT;	//current CPU temperature in °C
	AverageFrequency 										:	UDINT;		//average CPU frequency
	AverageUsage	 										:	UINT;		//average CPU usage in %
	AverageTemperature										:	INT;		//average CPU temperature in °C
	Count													:	INT; 		//number of CPUs
	ErrorGrp												:	E_MDP_ErrGroup := eMDP_Err_NoError;
END_VAR
VAR
	idx														:	INT := 1;
	MDP_ScanModules											:	FB_MDP_ScanModules := ( nModuleType 	:= eMDP_ModT_CPU , iModIdx		:= 0);
	MDP_Read												: 	FB_MDP_ReadModuleContent;
	SplitErrorId											:	FB_MDP_SplitErrorID;
	DstBuf													:	ARRAY[0..13] OF BYTE;
END_VAR

(* Read CPU Information 						V1.0		*)
(************************************************************)

(* Start Read ***********************************************)
	IF Execute
		AND state = 0
	THEN
		MEMSET(ADR(Frequency),0,SIZEOF(Frequency));
		MEMSET(ADR(Usage),0,SIZEOF(Usage));
		MEMSET(ADR(Temperature),0,SIZEOF(Temperature));
		AverageFrequency									:= 0;
		AverageUsage										:= 0;
		AverageTemperature									:= 0;
		Count												:= 0;
		Busy												:= TRUE;
		Done												:= FALSE;
		Error												:= FALSE;
		ErrorId												:= 0;
		ErrorGrp											:= eMDP_Err_NoError;
		MDP_Read(bExecute := FALSE);
		MDP_ScanModules(
			bExecute		:= FALSE,
			nModuleType		:= eMDP_ModT_CPU,
			iModIdx			:= 0,
			tTimeout		:= timeout,
			sAmsNetId		:= AmsNetId,
			bBusy			=> ,
			bError			=> ,
			nErrID			=> ,
			nDynModuleId	=> ,
			iModuleTypeCount=> ,
			iModuleCount	=> );
			
		MDP_ScanModules(bExecute		:= TRUE);		
		state												:= 1 ;
		
	ELSIF NOT Execute
		AND State = 99
	THEN
		state												:= 0;
		Busy												:= FALSE;
		Done												:= FALSE;
		Error												:= FALSE;
		ErrorId												:= 0;
		ErrorGrp											:= eMDP_Err_NoError;
	END_IF


	CASE state OF
	0:
		;
	1:
		MDP_ScanModules();
		IF NOT MDP_ScanModules.bBusy
		THEN
			IF MDP_ScanModules.bError
			THEN
				Busy										:= FALSE;
				Error										:= TRUE;
				SplitErrorId(
					nErrID		:= MDP_ScanModules.nErrID,
					eErrGroup	=> ErrorGrp ,
					nErrCode	=> ErrorId);
				state										:= 99;
				MDP_ScanModules(bExecute := FALSE);
			ELSE
				Count										:= MDP_ScanModules.iModuleTypeCount;
				MDP_Read.stMDP_DynAddr.nArea				:= 16#8;
				MDP_Read.stMDP_DynAddr.nModuleId			:= MDP_ScanModules.nDynModuleId;
				MDP_Read.stMDP_DynAddr.nSubIdx				:= 0;
				MDP_Read.stMDP_DynAddr.nTableId				:= 1;
				MDP_Read(bExecute := FALSE);
				idx											:= 1;
				IF Count = 0
				THEN
					Busy									:= FALSE;
					Error									:= TRUE;
					ErrorId									:= MDP_Read.nErrID;
					state									:= 99;
				ELSE
					MDP_Read(
						bExecute		:= TRUE,
						stMDP_DynAddr	:= ,
						iSubIdxCount	:= 4,
						pDstBuf			:= ADR(DstBuf),
						cbDstBufLen		:= SIZEOF(DstBuf),
						tTimeout		:= timeout,
						sAmsNetId		:= AmsNetId,
						bBusy			=> ,
						bError			=> ,
						nErrID			=> ,
						iErrPos			=> ,
						arrStartIdx		=> );
					state									:= 2;
				END_IF
			END_IF

		END_IF

	2:
		MDP_Read( pDstBuf := ADR(DstBuf), cbDstBufLen := SIZEOF(DstBuf));
		
		IF NOT MDP_Read.bBusy
		THEN
			IF MDP_Read.bError AND MDP_Read.iErrPos <> 4 AND MDP_Read.bExecute
			THEN
				Busy										:= FALSE;
				Error										:= TRUE;
				SplitErrorId(
					nErrID		:= MDP_Read.nErrID,
					eErrGroup	=> ErrorGrp ,
					nErrCode	=> ErrorId);
				state										:= 99;
				MDP_Read(bExecute := FALSE);
			ELSE
				(* copy freq *)
				IF MDP_Read.arrStartIdx[1] >= 0
				THEN
					MEMCPY( ADR(Frequency[idx]) , ADR(DstBuf[MDP_Read.arrStartIdx[1]]) , SIZEOF(Frequency[idx]) );
				END_IF
				(* copy usage *)
				IF MDP_Read.arrStartIdx[2] <> 0
				THEN
					MEMCPY(ADR(Usage[idx]) , ADR(DstBuf[MDP_Read.arrStartIdx[2]]) , SIZEOF(Usage[idx]) );
				END_IF
				(* copy temp in availible *)
				IF MDP_Read.arrStartIdx[3] <> 0
				THEN
					MEMCPY(ADR(Temperature[idx]) , ADR(DstBuf[MDP_Read.arrStartIdx[3]]) , SIZEOF(Temperature[idx]) ) ;
				END_IF

				MDP_Read(bExecute := FALSE);
				MDP_Read.stMDP_DynAddr.nModuleId := MDP_Read.stMDP_DynAddr.nModuleId + 1;
				
